Universal Robots PolyScope program: ratbit.urp

Program ratbit (installation=default directory=/programs createdIn=5.11.9.1010452 lastSavedIn=5.11.9.1010452 robotSerialNumber=20225200364)
Calibrated DH parameters: a=[0.00002, -0.569483, -0.54992, -0.00001, -0.000036, 0]; d=[0.180894, -146.691669, 192.918669, -46.053088, 0.119778, 0.115602]; alpha=[1.571425, -0.001534, 0.003359, 1.568739, -1.571477, 0]; deltaTheta=[0, 0.376258, -0.101074, -0.275185, -0.000002, 0]
Robot Program (runOnlyOnce=false)
  Script file /programs/Fuk_Rabbit_01D_newpath.script
    | def Machining1():
    |   # Global parameters:
    |   global speed_ms    = 0.300
    |   global speed_rads  = 0.750
    |   global accel_mss   = 3.000
    |   global accel_radss = 1.200
    |   global blend_radius_m = 0.001
    | 
    |   #--------------------------
    |   # Add any default subprograms here
    |   # For example, to drive a gripper as a program call:
    |   # def Gripper_Open():
    |   #   ...
    |   # end
    |   #
    |   # Example to drive a spray gun:
    |   def SprayOn(value):
    |     # use the value as an output:
    |     DO_SPRAY = 5
    |     if value == 0:
    |       set_standard_digital_out(DO_SPRAY, False)
    |     else:
    |       set_standard_digital_out(DO_SPRAY, True)
    |     end
    |   end
    |   #
    |   # Example to move an external axis
    |   def MoveAxis(value):
    |     # use the value as an output:
    |     DO_AXIS_1 = 1
    |     DI_AXIS_1 = 1
    |     if value <= 0:
    |       set_standard_digital_out(DO_AXIS_1, False)
    | 
    |       # Wait for digital input to change state
    |       #while (get_standard_digital_in(DI_AXIS_1) != False):
    |       #  sync()
    |       #end
    |     else:
    |       set_standard_digital_out(DO_AXIS_1, True)
    | 
    |       # Wait for digital input to change state
    |       #while (get_standard_digital_in(DI_AXIS_1) != True):
    |       #  sync()
    |       #end
    |     end
    |   end
    |   #--------------------------
    | 
    | 
    |   # Main program:
    |   # Program generated by RoboDK v5.4.3 for UR10e on 17/01/2023 09:30:10
    |   # Using nominal kinematics.
    |   blend_radius_m = 0.000
    |   speed_ms    = 1.000
    |   # set_reference(p[0.516600, -0.149080, 0.000000, 0.000000, 0.000000, 1.570796])
    |   set_tcp(p[0.000000, 0.000000, 0.25200, 0.000000, 0.000000, 0.000000])
    |   # Show Ballpen_2
    |   movej([0.053070, -1.824654, -1.998873, -4.030436, -1.570796, -1.517726],accel_radss,speed_rads,0,0)
    |   movel(p[0.486123, -0.148573, 0.015000, 0.000000, -3.141593, 0.000000],accel_mss,speed_ms,0,0)
    |   speed_ms    = 1.000
    |   movel(p[0.486123, -0.148573, 0.003000, 0.000000, -3.141593, 0.000000],accel_mss,speed_ms,0,blend_radius_m)
    |   speed_ms    = 0.050
    |   movel(p[0.486123, -0.148573, -0.000100, 0.000000, -3.141593, 0.000000],accel_mss,speed_ms,0,blend_radius_m)
    |   speed_ms    = 0.083
    |   movel(p[0.485906, -0.148799, -0.000100, 0.000000, -3.141593, 0.000000],accel_mss,speed_ms,0,0.000)
    |   movel(p[0.485689, -0.149025, -0.000100, 0.000000, -3.141593, 0.000000],accel_mss,speed_ms,0,0.000)
    |   movel(p[0.485511, -0.149199, -0.000100, 0.000000, -3.141593, 0.000000],accel_mss,speed_ms,0,0.000)
    |   movel(p[0.485335, -0.149346, -0.000100, 0.000000, -3.141593, 0.000000],accel_mss,speed_ms,0,0.000)
    |   movel(p[0.485182, -0.149454, -0.000100, 0.000000, -3.141593, 0.000000],accel_mss,speed_ms,0,0.000)
    |   movel(p[0.484988, -0.149437, -0.000100, 0.000000, -3.141593, 0.000000],accel_mss,speed_ms,0,0.000)
    |   movel(p[0.484142, -0.148632, -0.000100, 0.000000, -3.141593, 0.000000],accel_mss,speed_ms,0,blend_radius_m)
    |   movel(p[0.483183, -0.147699, -0.000100, 0.000000, -3.141593, 0.000000],accel_mss,speed_ms,0,blend_radius_m)
    |   movel(p[0.482074, -0.146592, -0.000100, 0.000000, -3.141593, 0.000000],accel_mss,speed_ms,0,blend_radius_m)
    |   movel(p[0.480976, -0.145473, -0.000100, 0.000000, -3.141593, 0.000000],accel_mss,speed_ms,0,blend_radius_m)
    |   movel(p[0.480046, -0.144505, -0.000100, 0.000000, -3.141593, 0.000000],accel_mss,speed_ms,0,blend_radius_m)
    |   movel(p[0.479240, -0.143652, -0.000100, 0.000000, -3.141593, 0.000000],accel_mss,speed_ms,0,blend_radius_m)
    |   movel(p[0.479187, -0.143544, -0.000100, 0.000000, -3.141593, 0.000000],accel_mss,speed_ms,0,0.000)
    |   movel(p[0.479279, -0.143263, -0.000100, 0.000000, -3.141593, 0.000000],accel_mss,speed_ms,0,0.000)
    |   movel(p[0.480734, -0.141843, -0.000100, 0.000000, -3.141593, 0.000000],accel_mss,speed_ms,0,blend_radius_m)
    |   movel(p[0.482145, -0.140509, -0.000100, 0.000000, -3.141593, 0.000000],accel_mss,speed_ms,0,blend_radius_m)
    |   movel(p[0.482666, -0.140186, -0.000100, 0.000000, -3.141593, 0.000000],accel_mss,speed_ms,0,blend_radius_m)
    |   movel(p[0.483571, -0.140040, -0.000100, 0.000000, -3.141593, 0.000000],accel_mss,speed_ms,0,blend_radius_m)
    |   movel(p[0.484504, -0.140251, -0.000100, 0.000000, -3.141593, 0.000000],accel_mss,speed_ms,0,blend_radius_m)
    |   movel(p[0.485320, -0.140784, -0.000100, 0.000000, -3.141593, 0.000000],accel_mss,speed_ms,0,blend_radius_m)
    |   movel(p[0.485889, -0.141559, -0.000100, 0.000000, -3.141593, 0.000000],accel_mss,speed_ms,0,blend_radius_m)
    |   movel(p[0.486167, -0.142427, -0.000100, 0.000000, -3.141593, 0.000000],accel_mss,speed_ms,0,blend_radius_m)
    |   movel(p[0.486122, -0.143201, -0.000100, 0.000000, -3.141593, 0.000000],accel_mss,speed_ms,0,blend_radius_m)
    |   movel(p[0.485720, -0.144015, -0.000100, 0.000000, -3.141593, 0.000000],accel_mss,speed_ms,0,blend_radius_m)
    |   movel(p[0.484872, -0.145041, -0.000100, 0.000000, -3.141593, 0.000000],accel_mss,speed_ms,0,blend_radius_m)
    |   movel(p[0.484523, -0.145430, -0.000100, 0.000000, -3.141593, 0.000000],accel_mss,speed_ms,0,blend_radius_m)
    |   movel(p[0.484229, -0.145788, -0.000100, 0.000000, -3.141593, 0.000000],accel_mss,speed_ms,0,0.000)
    |   movel(p[0.483998, -0.146094, -0.000100, 0.000000, -3.141593, 0.000000],accel_mss,speed_ms,0,0.000)
    |   movel(p[0.483961, -0.146209, -0.000100, 0.000000, -3.141593, 0.000000],accel_mss,speed_ms,0,0.000)
    |   movel(p[0.484001, -0.146324, -0.000100, 0.000000, -3.141593, 0.000000],accel_mss,speed_ms,0,0.000)
    |   movel(p[0.484278, -0.146661, -0.000100, 0.000000, -3.141593, 0.000000],accel_mss,speed_ms,0,0.000)
    |   movel(p[0.484628, -0.147054, -0.000100, 0.000000, -3.141593, 0.000000],accel_mss,speed_ms,0,blend_radius_m)
    |   movel(p[0.485042, -0.147484, -0.000100, 0.000000, -3.141593, 0.000000],accel_mss,speed_ms,0,blend_radius_m)
    |   movel(p[0.485582, -0.148028, -0.000100, 0.000000, -3.141593, 0.000000],accel_mss,speed_ms,0,blend_radius_m)
    |   movel(p[0.486123, -0.148573, -0.000100, 0.000000, -3.141593, 0.000000],accel_mss,speed_ms,0,blend_radius_m)
    |   speed_ms    = 0.050
    |   movel(p[0.486123, -0.148573, 0.003000, 0.000000, -3.141593, 0.000000],accel_mss,speed_ms,0,blend_radius_m)
    |   speed_ms    = 1.000
    |   movel(p[0.486123, -0.148573, 0.015000, 0.000000, -3.141593, 0.000000],accel_mss,speed_ms,0,blend_radius_m)
    |   movel(p[0.483124, -0.144911, 0.015000, 0.000000, -3.141593, 0.000000],accel_mss,speed_ms,0,blend_radius_m)
    |   movel(p[0.483124, -0.144911, 0.003000, 0.000000, -3.141593, 0.000000],accel_mss,speed_ms,0,blend_radius_m)
    |   speed_ms    = 0.050
    |   movel(p[0.483124, -0.144911, -0.000100, 0.000000, -3.141593, 0.000000],accel_mss,speed_ms,0,blend_radius_m)
    |   speed_ms    = 0.083
    |   movel(p[0.482775, -0.145021, -0.000100, 0.000000, -3.141593, 0.000000],accel_mss,speed_ms,0,0.000)
    |   movel(p[0.482418, -0.144857, -0.000100, 0.000000, -3.141593, 0.000000],accel_mss,speed_ms,0,0.000)
    |   movel(p[0.481726, -0.144152, -0.000100, 0.000000, -3.141593, 0.000000],accel_mss,speed_ms,0,blend_radius_m)
    |   movel(p[0.481290, -0.143631, -0.000100, 0.000000, -3.141593, 0.000000],accel_mss,speed_ms,0,blend_radius_m)
    |   movel(p[0.481235, -0.143353, -0.000100, 0.000000, -3.141593, 0.000000],accel_mss,speed_ms,0,0.000)
    |   movel(p[0.481407, -0.143059, -0.000100, 0.000000, -3.141593, 0.000000],accel_mss,speed_ms,0,0.000)
    |   movel(p[0.482217, -0.142290, -0.000100, 0.000000, -3.141593, 0.000000],accel_mss,speed_ms,0,blend_radius_m)
    |   movel(p[0.482465, -0.142075, -0.000100, 0.000000, -3.141593, 0.000000],accel_mss,speed_ms,0,0.000)
    |   movel(p[0.482730, -0.141875, -0.000100, 0.000000, -3.141593, 0.000000],accel_mss,speed_ms,0,0.000)
    |   movel(p[0.482975, -0.141713, -0.000100, 0.000000, -3.141593, 0.000000],accel_mss,speed_ms,0,0.000)
    |   movel(p[0.483149, -0.141630, -0.000100, 0.000000, -3.141593, 0.000000],accel_mss,speed_ms,0,0.000)
    |   movel(p[0.483717, -0.141623, -0.000100, 0.000000, -3.141593, 0.000000],accel_mss,speed_ms,0,blend_radius_m)
    |   movel(p[0.484256, -0.141955, -0.000100, 0.000000, -3.141593, 0.000000],accel_mss,speed_ms,0,blend_radius_m)
    |   movel(p[0.484596, -0.142514, -0.000100, 0.000000, -3.141593, 0.000000],accel_mss,speed_ms,0,blend_radius_m)
    |   movel(p[0.484618, -0.143123, -0.000100, 0.000000, -3.141593, 0.000000],accel_mss,speed_ms,0,blend_radius_m)
    |   movel(p[0.484529, -0.143332, -0.000100, 0.000000, -3.141593, 0.000000],accel_mss,speed_ms,0,0.000)
    |   movel(p[0.484314, -0.143650, -0.000100, 0.000000, -3.141593, 0.000000],accel_mss,speed_ms,0,0.000)
    |   movel(p[0.484037, -0.144003, -0.000100, 0.000000, -3.141593, 0.000000],accel_mss,speed_ms,0,0.000)
    |   movel(p[0.483729, -0.144344, -0.000100, 0.000000, -3.141593, 0.000000],accel_mss,speed_ms,0,0.000)
    |   movel(p[0.483124, -0.144911, -0.000100, 0.000000, -3.141593, 0.000000],accel_mss,speed_ms,0,blend_radius_m)
    |   speed_ms    = 0.050
    |   movel(p[0.483124, -0.144911, 0.003000, 0.000000, -3.141593, 0.000000],accel_mss,speed_ms,0,blend_radius_m)
    |   speed_ms    = 1.000
    |   movel(p[0.483124, -0.144911, 0.015000, 0.000000, -3.141593, 0.000000],accel_mss,speed_ms,0,blend_radius_m)
    |   movel(p[0.487811, -0.141414, 0.015000, 0.000000, -3.141593, 0.000000],accel_mss,speed_ms,0,blend_radius_m)
    |   movel(p[0.487811, -0.141414, 0.003000, 0.000000, -3.141593, 0.000000],accel_mss,speed_ms,0,blend_radius_m)
    |   speed_ms    = 0.050
    |   movel(p[0.487811, -0.141414, -0.000100, 0.000000, -3.141593, 0.000000],accel_mss,speed_ms,0,blend_radius_m)
    |   speed_ms    = 0.083
    |   movel(p[0.487491, -0.140892, -0.000100, 0.000000, -3.141593, 0.000000],accel_mss,speed_ms,0,blend_radius_m)
    |   movel(p[0.487400, -0.140626, -0.000100, 0.000000, -3.141593, 0.000000],accel_mss,speed_ms,0,0.000)
    |   movel(p[0.487339, -0.140285, -0.000100, 0.000000, -3.141593, 0.000000],accel_mss,speed_ms,0,0.000)
    |   movel(p[0.487307, -0.139892, -0.000100, 0.000000, -3.141593, 0.000000],accel_mss,speed_ms,0,0.000)
    |   movel(p[0.487310, -0.139469, -0.000100, 0.000000, -3.141593, 0.000000],accel_mss,speed_ms,0,0.000)
    |   movel(p[0.487439, -0.138661, -0.000100, 0.000000, -3.141593, 0.000000],accel_mss,speed_ms,0,blend_radius_m)
    |   movel(p[0.487749, -0.137963, -0.000100, 0.000000, -3.141593, 0.000000],accel_mss,speed_ms,0,blend_radius_m)
    |   movel(p[0.488242, -0.137381, -0.000100, 0.000000, -3.141593, 0.000000],accel_mss,speed_ms,0,blend_radius_m)
    |   movel(p[0.488911, -0.136916, -0.000100, 0.000000, -3.141593, 0.000000],accel_mss,speed_ms,0,blend_radius_m)
    |   movel(p[0.489677, -0.136642, -0.000100, 0.000000, -3.141593, 0.000000],accel_mss,speed_ms,0,blend_radius_m)
    |   movel(p[0.490526, -0.136585, -0.000100, 0.000000, -3.141593, 0.000000],accel_mss,speed_ms,0,blend_radius_m)
    |   movel(p[0.491362, -0.136747, -0.000100, 0.000000, -3.141593, 0.000000],accel_mss,speed_ms,0,blend_radius_m)
    |   movel(p[0.492092, -0.137115, -0.000100, 0.000000, -3.141593, 0.000000],accel_mss,speed_ms,0,blend_radius_m)
    |   movel(p[0.492654, -0.137612, -0.000100, 0.000000, -3.141593, 0.000000],accel_mss,speed_ms,0,blend_radius_m)
    |   movel(p[0.493144, -0.138258, -0.000100, 0.000000, -3.141593, 0.000000],accel_mss,speed_ms,0,blend_radius_m)
    |   movel(p[0.493503, -0.138962, -0.000100, 0.000000, -3.141593, 0.000000],accel_mss,speed_ms,0,blend_radius_m)
    |   movel(p[0.493671, -0.139629, -0.000100, 0.000000, -3.141593, 0.000000],accel_mss,speed_ms,0,blend_radius_m)
    |   movel(p[0.493430, -0.141150, -0.000100, 0.000000, -3.141593, 0.000000],accel_mss,speed_ms,0,blend_radius_m)
    |   movel(p[0.492438, -0.142384, -0.000100, 0.000000, -3.141593, 0.000000],accel_mss,speed_ms,0,blend_radius_m)
    |   movel(p[0.490977, -0.142992, -0.000100, 0.000000, -3.141593, 0.000000],accel_mss,speed_ms,0,blend_radius_m)
    |   movel(p[0.489451, -0.142800, -0.000100, 0.000000, -3.141593, 0.000000],accel_mss,speed_ms,0,blend_radius_m)
    |   movel(p[0.488923, -0.142496, -0.000100, 0.000000, -3.141593, 0.000000],accel_mss,speed_ms,0,blend_radius_m)
    |   movel(p[0.488334, -0.141990, -0.000100, 0.000000, -3.141593, 0.000000],accel_mss,speed_ms,0,blend_radius_m)
    |   movel(p[0.487811, -0.141414, -0.000100, 0.000000, -3.141593, 0.000000],accel_mss,speed_ms,0,blend_radius_m)
    |   speed_ms    = 0.050
    |   movel(p[0.487811, -0.141414, 0.003000, 0.000000, -3.141593, 0.000000],accel_mss,speed_ms,0,blend_radius_m)
    |   speed_ms    = 1.000
    |   movel(p[0.487811, -0.141414, 0.015000, 0.000000, -3.141593, 0.000000],accel_mss,speed_ms,0,blend_radius_m)
    |   movel(p[0.489267, -0.140905, 0.015000, 0.000000, -3.141593, 0.000000],accel_mss,speed_ms,0,blend_radius_m)
    |   movel(p[0.489267, -0.140905, 0.003000, 0.000000, -3.141593, 0.000000],accel_mss,speed_ms,0,blend_radius_m)
    |   speed_ms    = 0.050
    |   movel(p[0.489267, -0.140905, -0.000100, 0.000000, -3.141593, 0.000000],accel_mss,speed_ms,0,blend_radius_m)
    |   speed_ms    = 0.083
    |   movel(p[0.488764, -0.140201, -0.000100, 0.000000, -3.141593, 0.000000],accel_mss,speed_ms,0,blend_radius_m)
    |   movel(p[0.488534, -0.139500, -0.000100, 0.000000, -3.141593, 0.000000],accel_mss,speed_ms,0,blend_radius_m)
    |   movel(p[0.488593, -0.138851, -0.000100, 0.000000, -3.141593, 0.000000],accel_mss,speed_ms,0,blend_radius_m)
    |   movel(p[0.488924, -0.138290, -0.000100, 0.000000, -3.141593, 0.000000],accel_mss,speed_ms,0,blend_radius_m)
    |   movel(p[0.489534, -0.137898, -0.000100, 0.000000, -3.141593, 0.000000],accel_mss,speed_ms,0,blend_radius_m)
    |   movel(p[0.490256, -0.137841, -0.000100, 0.000000, -3.141593, 0.000000],accel_mss,speed_ms,0,blend_radius_m)
    |   movel(p[0.491020, -0.138140, -0.000100, 0.000000, -3.141593, 0.000000],accel_mss,speed_ms,0,blend_radius_m)
    |   movel(p[0.491739, -0.138764, -0.000100, 0.000000, -3.141593, 0.000000],accel_mss,speed_ms,0,blend_radius_m)
    |   movel(p[0.492146, -0.139301, -0.000100, 0.000000, -3.141593, 0.000000],accel_mss,speed_ms,0,blend_radius_m)
    |   movel(p[0.492374, -0.139794, -0.000100, 0.000000, -3.141593, 0.000000],accel_mss,speed_ms,0,blend_radius_m)
    |   movel(p[0.492436, -0.140272, -0.000100, 0.000000, -3.141593, 0.000000],accel_mss,speed_ms,0,0.000)
    |   movel(p[0.492345, -0.140761, -0.000100, 0.000000, -3.141593, 0.000000],accel_mss,speed_ms,0,0.000)
    |   movel(p[0.491847, -0.141407, -0.000100, 0.000000, -3.141593, 0.000000],accel_mss,speed_ms,0,blend_radius_m)
    |   movel(p[0.491027, -0.141679, -0.000100, 0.000000, -3.141593, 0.000000],accel_mss,speed_ms,0,blend_radius_m)
    |   movel(p[0.490083, -0.141499, -0.000100, 0.000000, -3.141593, 0.000000],accel_mss,speed_ms,0,blend_radius_m)
    |   movel(p[0.489267, -0.140905, -0.000100, 0.000000, -3.141593, 0.000000],accel_mss,speed_ms,0,blend_radius_m)
    |   speed_ms    = 0.050
    |   movel(p[0.489267, -0.140905, 0.003000, 0.000000, -3.141593, 0.000000],accel_mss,speed_ms,0,blend_radius_m)
    |   speed_ms    = 1.000
    |   movel(p[0.489267, -0.140905, 0.015000, 0.000000, -3.141593, 0.000000],accel_mss,speed_ms,0,blend_radius_m)
    |   movel(p[0.494074, -0.136704, 0.015000, 0.000000, -3.141593, 0.000000],accel_mss,speed_ms,0,blend_radius_m)
    |   movel(p[0.494074, -0.136704, 0.003000, 0.000000, -3.141593, 0.000000],accel_mss,speed_ms,0,blend_radius_m)
    |   speed_ms    = 0.050
    |   movel(p[0.494074, -0.136704, -0.000100, 0.000000, -3.141593, 0.000000],accel_mss,speed_ms,0,blend_radius_m)
    |   speed_ms    = 0.083
    |   movel(p[0.492928, -0.135570, -0.000100, 0.000000, -3.141593, 0.000000],accel_mss,speed_ms,0,blend_radius_m)
    |   movel(p[0.491447, -0.134091, -0.000100, 0.000000, -3.141593, 0.000000],accel_mss,speed_ms,0,blend_radius_m)
    |   movel(p[0.489967, -0.132612, -0.000100, 0.000000, -3.141593, 0.000000],accel_mss,speed_ms,0,blend_radius_m)
    |   movel(p[0.490207, -0.132364, -0.000100, 0.000000, -3.141593, 0.000000],accel_mss,speed_ms,0,0.000)
    |   movel(p[0.490447, -0.132117, -0.000100, 0.000000, -3.141593, 0.000000],accel_mss,speed_ms,0,0.000)
    |   movel(p[0.490686, -0.131869, -0.000100, 0.000000, -3.141593, 0.000000],accel_mss,speed_ms,0,0.000)
    |   movel(p[0.490926, -0.131622, -0.000100, 0.000000, -3.141593, 0.000000],accel_mss,speed_ms,0,0.000)
    |   movel(p[0.492410, -0.133104, -0.000100, 0.000000, -3.141593, 0.000000],accel_mss,speed_ms,0,blend_radius_m)
    |   movel(p[0.493894, -0.134586, -0.000100, 0.000000, -3.141593, 0.000000],accel_mss,speed_ms,0,blend_radius_m)
    |   movel(p[0.495031, -0.135733, -0.000100, 0.000000, -3.141593, 0.000000],accel_mss,speed_ms,0,blend_radius_m)
    |   movel(p[0.495989, -0.136721, -0.000100, 0.000000, -3.141593, 0.000000],accel_mss,speed_ms,0,blend_radius_m)
    |   movel(p[0.496823, -0.137596, -0.000100, 0.000000, -3.141593, 0.000000],accel_mss,speed_ms,0,blend_radius_m)
    |   movel(p[0.496861, -0.137692, -0.000100, 0.000000, -3.141593, 0.000000],accel_mss,speed_ms,0,0.000)
    |   movel(p[0.496796, -0.137879, -0.000100, 0.000000, -3.141593, 0.000000],accel_mss,speed_ms,0,0.000)
    |   movel(p[0.496527, -0.138185, -0.000100, 0.000000, -3.141593, 0.000000],accel_mss,speed_ms,0,0.000)
    |   movel(p[0.496230, -0.138462, -0.000100, 0.000000, -3.141593, 0.000000],accel_mss,speed_ms,0,0.000)
    |   movel(p[0.496049, -0.138528, -0.000100, 0.000000, -3.141593, 0.000000],accel_mss,speed_ms,0,0.000)
    |   movel(p[0.495941, -0.138486, -0.000100, 0.000000, -3.141593, 0.000000],accel_mss,speed_ms,0,0.000)
    |   movel(p[0.495066, -0.137659, -0.000100, 0.000000, -3.141593, 0.000000],accel_mss,speed_ms,0,blend_radius_m)
    |   movel(p[0.494074, -0.136704, -0.000100, 0.000000, -3.141593, 0.000000],accel_mss,speed_ms,0,blend_radius_m)
    |   speed_ms    = 0.050
    |   movel(p[0.494074, -0.136704, 0.003000, 0.000000, -3.141593, 0.000000],accel_mss,speed_ms,0,blend_radius_m)
    |   speed_ms    = 1.000
    |   movel(p[0.494074, -0.136704, 0.015000, 0.000000, -3.141593, 0.000000],accel_mss,speed_ms,0,blend_radius_m)
    |   movel(p[0.495341, -0.133290, 0.015000, 0.000000, -3.141593, 0.000000],accel_mss,speed_ms,0,blend_radius_m)
    |   movel(p[0.495341, -0.133290, 0.003000, 0.000000, -3.141593, 0.000000],accel_mss,speed_ms,0,blend_radius_m)
    |   speed_ms    = 0.050
    |   movel(p[0.495341, -0.133290, -0.000100, 0.000000, -3.141593, 0.000000],accel_mss,speed_ms,0,blend_radius_m)
    |   speed_ms    = 0.083
    |   movel(p[0.494409, -0.132847, -0.000100, 0.000000, -3.141593, 0.000000],accel_mss,speed_ms,0,blend_radius_m)
    |   movel(p[0.493590, -0.132450, -0.000100, 0.000000, -3.141593, 0.000000],accel_mss,speed_ms,0,blend_radius_m)
    |   movel(p[0.493631, -0.132230, -0.000100, 0.000000, -3.141593, 0.000000],accel_mss,speed_ms,0,0.000)
    |   movel(p[0.493992, -0.131876, -0.000100, 0.000000, -3.141593, 0.000000],accel_mss,speed_ms,0,blend_radius_m)
    |   movel(p[0.494374, -0.131546, -0.000100, 0.000000, -3.141593, 0.000000],accel_mss,speed_ms,0,blend_radius_m)
    |   movel(p[0.494564, -0.131478, -0.000100, 0.000000, -3.141593, 0.000000],accel_mss,speed_ms,0,0.000)
    |   movel(p[0.494698, -0.131507, -0.000100, 0.000000, -3.141593, 0.000000],accel_mss,speed_ms,0,0.000)
    |   movel(p[0.495213, -0.131743, -0.000100, 0.000000, -3.141593, 0.000000],accel_mss,speed_ms,0,blend_radius_m)
    |   movel(p[0.495818, -0.132033, -0.000100, 0.000000, -3.141593, 0.000000],accel_mss,speed_ms,0,blend_radius_m)
    |   movel(p[0.496498, -0.132378, -0.000100, 0.000000, -3.141593, 0.000000],accel_mss,speed_ms,0,blend_radius_m)
    |   movel(p[0.497622, -0.132946, -0.000100, 0.000000, -3.141593, 0.000000],accel_mss,speed_ms,0,blend_radius_m)
    |   movel(p[0.498224, -0.133197, -0.000100, 0.000000, -3.141593, 0.000000],accel_mss,speed_ms,0,blend_radius_m)
    |   movel(p[0.498543, -0.133247, -0.000100, 0.000000, -3.141593, 0.000000],accel_mss,speed_ms,0,0.000)
    |   movel(p[0.498661, -0.133126, -0.000100, 0.000000, -3.141593, 0.000000],accel_mss,speed_ms,0,0.000)
    |   movel(p[0.498637, -0.133018, -0.000100, 0.000000, -3.141593, 0.000000],accel_mss,speed_ms,0,0.000)
    |   movel(p[0.498377, -0.132453, -0.000100, 0.000000, -3.141593, 0.000000],accel_mss,speed_ms,0,blend_radius_m)
    |   movel(p[0.498065, -0.131796, -0.000100, 0.000000, -3.141593, 0.000000],accel_mss,speed_ms,0,blend_radius_m)
    |   movel(p[0.497695, -0.131047, -0.000100, 0.000000, -3.141593, 0.000000],accel_mss,speed_ms,0,blend_radius_m)
    |   movel(p[0.497212, -0.130083, -0.000100, 0.000000, -3.141593, 0.000000],accel_mss,speed_ms,0,blend_radius_m)
    |   movel(p[0.496729, -0.129119, -0.000100, 0.000000, -3.141593, 0.000000],accel_mss,speed_ms,0,blend_radius_m)
    |   movel(p[0.496985, -0.128871, -0.000100, 0.000000, -3.141593, 0.000000],accel_mss,speed_ms,0,0.000)
    |   movel(p[0.497241, -0.128624, -0.000100, 0.000000, -3.141593, 0.000000],accel_mss,speed_ms,0,0.000)
    |   movel(p[0.497497, -0.128376, -0.000100, 0.000000, -3.141593, 0.000000],accel_mss,speed_ms,0,0.000)
    |   movel(p[0.497752, -0.128128, -0.000100, 0.000000, -3.141593, 0.000000],accel_mss,speed_ms,0,0.000)
    |   movel(p[0.498286, -0.129247, -0.000100, 0.000000, -3.141593, 0.000000],accel_mss,speed_ms,0,blend_radius_m)
    |   movel(p[0.498819, -0.130366, -0.000100, 0.000000, -3.141593, 0.000000],accel_mss,speed_ms,0,blend_radius_m)
    |   # Splitting circular movement in 4 (instruction 203:MoveC 176)
    |   movel(p[0.499281, -0.131340, -0.000100, 0.000000, -3.141593, 0.000000],accel_mss,speed_ms,0,blend_radius_m)
    |   movel(p[0.499741, -0.132315, -0.000100, 0.000000, -3.141593, 0.000000],accel_mss,speed_ms,0,blend_radius_m)
    |   movel(p[0.500197, -0.133292, -0.000100, 0.000000, -3.141593, 0.000000],accel_mss,speed_ms,0,blend_radius_m)
    |   movel(p[0.500650, -0.134270, -0.000100, 0.000000, -3.141593, 0.000000],accel_mss,speed_ms,0,blend_radius_m)
    |   movel(p[0.501168, -0.135720, -0.000100, 0.000000, -3.141593, 0.000000],accel_mss,speed_ms,0,blend_radius_m)
    |   movel(p[0.501150, -0.136625, -0.000100, 0.000000, -3.141593, 0.000000],accel_mss,speed_ms,0,blend_radius_m)
    |   movel(p[0.500669, -0.137478, -0.000100, 0.000000, -3.141593, 0.000000],accel_mss,speed_ms,0,blend_radius_m)
    |   movel(p[0.500264, -0.137878, -0.000100, 0.000000, -3.141593, 0.000000],accel_mss,speed_ms,0,blend_radius_m)
    |   movel(p[0.499962, -0.138042, -0.000100, 0.000000, -3.141593, 0.000000],accel_mss,speed_ms,0,0.000)
    |   movel(p[0.499687, -0.138024, -0.000100, 0.000000, -3.141593, 0.000000],accel_mss,speed_ms,0,0.000)
    |   movel(p[0.499389, -0.137833, -0.000100, 0.000000, -3.141593, 0.000000],accel_mss,speed_ms,0,0.000)
    |   movel(p[0.499240, -0.137674, -0.000100, 0.000000, -3.141593, 0.000000],accel_mss,speed_ms,0,0.000)
    |   movel(p[0.499210, -0.137558, -0.000100, 0.000000, -3.141593, 0.000000],accel_mss,speed_ms,0,0.000)
    |   movel(p[0.499270, -0.137421, -0.000100, 0.000000, -3.141593, 0.000000],accel_mss,speed_ms,0,0.000)
    |   movel(p[0.499505, -0.137128, -0.000100, 0.000000, -3.141593, 0.000000],accel_mss,speed_ms,0,0.000)
    |   movel(p[0.499701, -0.136864, -0.000100, 0.000000, -3.141593, 0.000000],accel_mss,speed_ms,0,0.000)
    |   movel(p[0.499803, -0.136643, -0.000100, 0.000000, -3.141593, 0.000000],accel_mss,speed_ms,0,0.000)
    |   movel(p[0.499836, -0.136403, -0.000100, 0.000000, -3.141593, 0.000000],accel_mss,speed_ms,0,0.000)
    |   movel(p[0.499813, -0.136078, -0.000100, 0.000000, -3.141593, 0.000000],accel_mss,speed_ms,0,0.000)
    |   movel(p[0.499768, -0.135838, -0.000100, 0.000000, -3.141593, 0.000000],accel_mss,speed_ms,0,0.000)
    |   movel(p[0.499699, -0.135606, -0.000100, 0.000000, -3.141593, 0.000000],accel_mss,speed_ms,0,0.000)
    |   movel(p[0.499617, -0.135412, -0.000100, 0.000000, -3.141593, 0.000000],accel_mss,speed_ms,0,0.000)
    |   movel(p[0.499535, -0.135302, -0.000100, 0.000000, -3.141593, 0.000000],accel_mss,speed_ms,0,0.000)
    |   movel(p[0.499374, -0.135190, -0.000100, 0.000000, -3.141593, 0.000000],accel_mss,speed_ms,0,0.000)
    |   movel(p[0.498546, -0.134784, -0.000100, 0.000000, -3.141593, 0.000000],accel_mss,speed_ms,0,blend_radius_m)
    |   movel(p[0.497569, -0.134318, -0.000100, 0.000000, -3.141593, 0.000000],accel_mss,speed_ms,0,blend_radius_m)
    |   movel(p[0.496448, -0.133801, -0.000100, 0.000000, -3.141593, 0.000000],accel_mss,speed_ms,0,blend_radius_m)
    |   movel(p[0.495341, -0.133290, -0.000100, 0.000000, -3.141593, 0.000000],accel_mss,speed_ms,0,blend_radius_m)
    |   speed_ms    = 0.050
    |   movel(p[0.495341, -0.133290, 0.003000, 0.000000, -3.141593, 0.000000],accel_mss,speed_ms,0,blend_radius_m)
    |   speed_ms    = 1.000
    |   movel(p[0.495341, -0.133290, 0.015000, 0.000000, -3.141593, 0.000000],accel_mss,speed_ms,0,blend_radius_m)
    |   movel(p[0.500261, -0.128751, 0.015000, 0.000000, -3.141593, 0.000000],accel_mss,speed_ms,0,blend_radius_m)
    |   movel(p[0.500261, -0.128751, 0.003000, 0.000000, -3.141593, 0.000000],accel_mss,speed_ms,0,blend_radius_m)
    |   speed_ms    = 0.050
    |   movel(p[0.500261, -0.128751, -0.000100, 0.000000, -3.141593, 0.000000],accel_mss,speed_ms,0,blend_radius_m)
    |   speed_ms    = 0.083
    |   movel(p[0.499327, -0.127855, -0.000100, 0.000000, -3.141593, 0.000000],accel_mss,speed_ms,0,blend_radius_m)
    |   movel(p[0.498163, -0.126713, -0.000100, 0.000000, -3.141593, 0.000000],accel_mss,speed_ms,0,blend_radius_m)
    |   movel(p[0.497000, -0.125570, -0.000100, 0.000000, -3.141593, 0.000000],accel_mss,speed_ms,0,blend_radius_m)
    |   movel(p[0.497263, -0.125306, -0.000100, 0.000000, -3.141593, 0.000000],accel_mss,speed_ms,0,0.000)
    |   movel(p[0.497526, -0.125043, -0.000100, 0.000000, -3.141593, 0.000000],accel_mss,speed_ms,0,0.000)
    |   movel(p[0.497790, -0.124780, -0.000100, 0.000000, -3.141593, 0.000000],accel_mss,speed_ms,0,0.000)
    |   movel(p[0.498053, -0.124516, -0.000100, 0.000000, -3.141593, 0.000000],accel_mss,speed_ms,0,0.000)
    |   movel(p[0.499161, -0.125608, -0.000100, 0.000000, -3.141593, 0.000000],accel_mss,speed_ms,0,blend_radius_m)
    |   movel(p[0.500269, -0.126699, -0.000100, 0.000000, -3.141593, 0.000000],accel_mss,speed_ms,0,blend_radius_m)
    |   movel(p[0.501231, -0.127626, -0.000100, 0.000000, -3.141593, 0.000000],accel_mss,speed_ms,0,blend_radius_m)
    |   movel(p[0.502013, -0.128332, -0.000100, 0.000000, -3.141593, 0.000000],accel_mss,speed_ms,0,blend_radius_m)
    |   movel(p[0.502632, -0.128847, -0.000100, 0.000000, -3.141593, 0.000000],accel_mss,speed_ms,0,blend_radius_m)
    |   movel(p[0.502914, -0.128986, -0.000100, 0.000000, -3.141593, 0.000000],accel_mss,speed_ms,0,0.000)
    |   movel(p[0.503793, -0.128942, -0.000100, 0.000000, -3.141593, 0.000000],accel_mss,speed_ms,0,blend_radius_m)
    |   movel(p[0.504622, -0.128423, -0.000100, 0.000000, -3.141593, 0.000000],accel_mss,speed_ms,0,blend_radius_m)
    |   movel(p[0.505149, -0.127606, -0.000100, 0.000000, -3.141593, 0.000000],accel_mss,speed_ms,0,blend_radius_m)
    |   movel(p[0.505195, -0.126738, -0.000100, 0.000000, -3.141593, 0.000000],accel_mss,speed_ms,0,blend_radius_m)
    |   movel(p[0.505072, -0.126494, -0.000100, 0.000000, -3.141593, 0.000000],accel_mss,speed_ms,0,0.000)
    |   movel(p[0.504490, -0.125812, -0.000100, 0.000000, -3.141593, 0.000000],accel_mss,speed_ms,0,blend_radius_m)
    |   movel(p[0.503761, -0.125006, -0.000100, 0.000000, -3.141593, 0.000000],accel_mss,speed_ms,0,blend_radius_m)
    |   movel(p[0.502900, -0.124107, -0.000100, 0.000000, -3.141593, 0.000000],accel_mss,speed_ms,0,blend_radius_m)
    |   movel(p[0.501801, -0.122987, -0.000100, 0.000000, -3.141593, 0.000000],accel_mss,speed_ms,0,blend_radius_m)
    |   movel(p[0.500703, -0.121867, -0.000100, 0.000000, -3.141593, 0.000000],accel_mss,speed_ms,0,blend_radius_m)
    |   movel(p[0.500966, -0.121603, -0.000100, 0.000000, -3.141593, 0.000000],accel_mss,speed_ms,0,0.000)
    |   movel(p[0.501229, -0.121340, -0.000100, 0.000000, -3.141593, 0.000000],accel_mss,speed_ms,0,0.000)
    |   movel(p[0.501492, -0.121077, -0.000100, 0.000000, -3.141593, 0.000000],accel_mss,speed_ms,0,0.000)
    |   movel(p[0.501755, -0.120814, -0.000100, 0.000000, -3.141593, 0.000000],accel_mss,speed_ms,0,0.000)
    |   movel(p[0.502877, -0.121961, -0.000100, 0.000000, -3.141593, 0.000000],accel_mss,speed_ms,0,blend_radius_m)
    |   movel(p[0.503998, -0.123109, -0.000100, 0.000000, -3.141593, 0.000000],accel_mss,speed_ms,0,blend_radius_m)
    |   movel(p[0.504876, -0.124028, -0.000100, 0.000000, -3.141593, 0.000000],accel_mss,speed_ms,0,blend_radius_m)
    |   movel(p[0.505659, -0.124891, -0.000100, 0.000000, -3.141593, 0.000000],accel_mss,speed_ms,0,blend_radius_m)
    |   movel(p[0.506293, -0.125628, -0.000100, 0.000000, -3.141593, 0.000000],accel_mss,speed_ms,0,blend_radius_m)
    |   movel(p[0.506501, -0.125951, -0.000100, 0.000000, -3.141593, 0.000000],accel_mss,speed_ms,0,0.000)
    |   movel(p[0.506729, -0.126810, -0.000100, 0.000000, -3.141593, 0.000000],accel_mss,speed_ms,0,blend_radius_m)
    |   movel(p[0.506629, -0.127680, -0.000100, 0.000000, -3.141593, 0.000000],accel_mss,speed_ms,0,blend_radius_m)
    |   movel(p[0.506186, -0.128560, -0.000100, 0.000000, -3.141593, 0.000000],accel_mss,speed_ms,0,blend_radius_m)
    |   movel(p[0.505401, -0.129448, -0.000100, 0.000000, -3.141593, 0.000000],accel_mss,speed_ms,0,blend_radius_m)
    |   movel(p[0.504548, -0.130125, -0.000100, 0.000000, -3.141593, 0.000000],accel_mss,speed_ms,0,blend_radius_m)
    |   movel(p[0.503759, -0.130489, -0.000100, 0.000000, -3.141593, 0.000000],accel_mss,speed_ms,0,blend_radius_m)
    |   movel(p[0.502984, -0.130560, -0.000100, 0.000000, -3.141593, 0.000000],accel_mss,speed_ms,0,blend_radius_m)
    |   movel(p[0.502178, -0.130360, -0.000100, 0.000000, -3.141593, 0.000000],accel_mss,speed_ms,0,blend_radius_m)
    |   movel(p[0.501865, -0.130170, -0.000100, 0.000000, -3.141593, 0.000000],accel_mss,speed_ms,0,0.000)
    |   movel(p[0.501127, -0.129537, -0.000100, 0.000000, -3.141593, 0.000000],accel_mss,speed_ms,0,blend_radius_m)
    |   movel(p[0.500261, -0.128751, -0.000100, 0.000000, -3.141593, 0.000000],accel_mss,speed_ms,0,blend_radius_m)
    |   speed_ms    = 0.050
    |   movel(p[0.500261, -0.128751, 0.003000, 0.000000, -3.141593, 0.000000],accel_mss,speed_ms,0,blend_radius_m)
    |   speed_ms    = 1.000
    |   movel(p[0.500261, -0.128751, 0.015000, 0.000000, -3.141593, 0.000000],accel_mss,speed_ms,0,blend_radius_m)
    |   movel(p[0.508525, -0.119968, 0.015000, 0.000000, -3.141593, 0.000000],accel_mss,speed_ms,0,blend_radius_m)
    |   movel(p[0.508525, -0.119968, 0.003000, 0.000000, -3.141593, 0.000000],accel_mss,speed_ms,0,blend_radius_m)
    |   speed_ms    = 0.050
    |   movel(p[0.508525, -0.119968, -0.000100, 0.000000, -3.141593, 0.000000],accel_mss,speed_ms,0,blend_radius_m)
    |   speed_ms    = 0.083
    |   movel(p[0.507044, -0.118488, -0.000100, 0.000000, -3.141593, 0.000000],accel_mss,speed_ms,0,blend_radius_m)
    |   movel(p[0.505562, -0.117007, -0.000100, 0.000000, -3.141593, 0.000000],accel_mss,speed_ms,0,blend_radius_m)
    |   movel(p[0.505825, -0.116745, -0.000100, 0.000000, -3.141593, 0.000000],accel_mss,speed_ms,0,0.000)
    |   movel(p[0.506088, -0.116482, -0.000100, 0.000000, -3.141593, 0.000000],accel_mss,speed_ms,0,0.000)
    |   movel(p[0.506350, -0.116219, -0.000100, 0.000000, -3.141593, 0.000000],accel_mss,speed_ms,0,0.000)
    |   movel(p[0.506613, -0.115956, -0.000100, 0.000000, -3.141593, 0.000000],accel_mss,speed_ms,0,0.000)
    |   movel(p[0.508118, -0.117462, -0.000100, 0.000000, -3.141593, 0.000000],accel_mss,speed_ms,0,blend_radius_m)
    |   movel(p[0.509624, -0.118967, -0.000100, 0.000000, -3.141593, 0.000000],accel_mss,speed_ms,0,blend_radius_m)
    |   movel(p[0.511129, -0.120472, -0.000100, 0.000000, -3.141593, 0.000000],accel_mss,speed_ms,0,blend_radius_m)
    |   movel(p[0.512634, -0.121978, -0.000100, 0.000000, -3.141593, 0.000000],accel_mss,speed_ms,0,blend_radius_m)
    |   movel(p[0.512434, -0.122215, -0.000100, 0.000000, -3.141593, 0.000000],accel_mss,speed_ms,0,0.000)
    |   movel(p[0.512234, -0.122453, -0.000100, 0.000000, -3.141593, 0.000000],accel_mss,speed_ms,0,0.000)
    |   movel(p[0.512068, -0.122635, -0.000100, 0.000000, -3.141593, 0.000000],accel_mss,speed_ms,0,0.000)
    |   movel(p[0.511901, -0.122789, -0.000100, 0.000000, -3.141593, 0.000000],accel_mss,speed_ms,0,0.000)
    |   movel(p[0.511752, -0.122901, -0.000100, 0.000000, -3.141593, 0.000000],accel_mss,speed_ms,0,0.000)
    |   movel(p[0.511545, -0.122882, -0.000100, 0.000000, -3.141593, 0.000000],accel_mss,speed_ms,0,0.000)
    |   movel(p[0.510669, -0.122059, -0.000100, 0.000000, -3.141593, 0.000000],accel_mss,speed_ms,0,blend_radius_m)
    |   movel(p[0.509674, -0.121103, -0.000100, 0.000000, -3.141593, 0.000000],accel_mss,speed_ms,0,blend_radius_m)
    |   movel(p[0.508525, -0.119968, -0.000100, 0.000000, -3.141593, 0.000000],accel_mss,speed_ms,0,blend_radius_m)
    |   speed_ms    = 0.050
    |   movel(p[0.508525, -0.119968, 0.003000, 0.000000, -3.141593, 0.000000],accel_mss,speed_ms,0,blend_radius_m)
    |   speed_ms    = 1.000
    |   movel(p[0.508525, -0.119968, 0.015000, 0.000000, -3.141593, 0.000000],accel_mss,speed_ms,0,blend_radius_m)
    |   movel(p[0.510708, -0.117772, 0.015000, 0.000000, -3.141593, 0.000000],accel_mss,speed_ms,0,blend_radius_m)
    |   movel(p[0.510708, -0.117772, 0.003000, 0.000000, -3.141593, 0.000000],accel_mss,speed_ms,0,blend_radius_m)
    |   speed_ms    = 0.050
    |   movel(p[0.510708, -0.117772, -0.000100, 0.000000, -3.141593, 0.000000],accel_mss,speed_ms,0,blend_radius_m)
    |   speed_ms    = 0.083
    |   movel(p[0.510076, -0.117035, -0.000100, 0.000000, -3.141593, 0.000000],accel_mss,speed_ms,0,blend_radius_m)
    |   movel(p[0.509614, -0.116286, -0.000100, 0.000000, -3.141593, 0.000000],accel_mss,speed_ms,0,blend_radius_m)
    |   movel(p[0.509278, -0.115433, -0.000100, 0.000000, -3.141593, 0.000000],accel_mss,speed_ms,0,blend_radius_m)
    |   movel(p[0.509157, -0.114640, -0.000100, 0.000000, -3.141593, 0.000000],accel_mss,speed_ms,0,blend_radius_m)
    |   movel(p[0.509248, -0.113863, -0.000100, 0.000000, -3.141593, 0.000000],accel_mss,speed_ms,0,blend_radius_m)
    |   movel(p[0.509549, -0.113059, -0.000100, 0.000000, -3.141593, 0.000000],accel_mss,speed_ms,0,blend_radius_m)
    |   movel(p[0.510352, -0.111920, -0.000100, 0.000000, -3.141593, 0.000000],accel_mss,speed_ms,0,blend_radius_m)
    |   movel(p[0.511427, -0.111135, -0.000100, 0.000000, -3.141593, 0.000000],accel_mss,speed_ms,0,blend_radius_m)
    |   movel(p[0.512614, -0.110814, -0.000100, 0.000000, -3.141593, 0.000000],accel_mss,speed_ms,0,blend_radius_m)
    |   movel(p[0.513747, -0.110998, -0.000100, 0.000000, -3.141593, 0.000000],accel_mss,speed_ms,0,blend_radius_m)
    |   movel(p[0.514084, -0.111150, -0.000100, 0.000000, -3.141593, 0.000000],accel_mss,speed_ms,0,0.000)
    |   movel(p[0.514178, -0.111247, -0.000100, 0.000000, -3.141593, 0.000000],accel_mss,speed_ms,0,0.000)
    |   movel(p[0.514179, -0.111374, -0.000100, 0.000000, -3.141593, 0.000000],accel_mss,speed_ms,0,0.000)
    |   movel(p[0.514043, -0.111664, -0.000100, 0.000000, -3.141593, 0.000000],accel_mss,speed_ms,0,0.000)
    |   movel(p[0.513816, -0.112030, -0.000100, 0.000000, -3.141593, 0.000000],accel_mss,speed_ms,0,0.000)
    |   movel(p[0.513591, -0.112219, -0.000100, 0.000000, -3.141593, 0.000000],accel_mss,speed_ms,0,0.000)
    |   movel(p[0.513275, -0.112311, -0.000100, 0.000000, -3.141593, 0.000000],accel_mss,speed_ms,0,0.000)
    |   movel(p[0.512696, -0.112344, -0.000100, 0.000000, -3.141593, 0.000000],accel_mss,speed_ms,0,blend_radius_m)
    |   movel(p[0.512355, -0.112368, -0.000100, 0.000000, -3.141593, 0.000000],accel_mss,speed_ms,0,0.000)
    |   movel(p[0.512032, -0.112428, -0.000100, 0.000000, -3.141593, 0.000000],accel_mss,speed_ms,0,0.000)
    |   movel(p[0.511749, -0.112517, -0.000100, 0.000000, -3.141593, 0.000000],accel_mss,speed_ms,0,0.000)
    |   movel(p[0.511531, -0.112630, -0.000100, 0.000000, -3.141593, 0.000000],accel_mss,speed_ms,0,0.000)
    |   movel(p[0.511128, -0.113018, -0.000100, 0.000000, -3.141593, 0.000000],accel_mss,speed_ms,0,blend_radius_m)
    |   movel(p[0.510791, -0.113595, -0.000100, 0.000000, -3.141593, 0.000000],accel_mss,speed_ms,0,blend_radius_m)
    |   movel(p[0.510582, -0.114217, -0.000100, 0.000000, -3.141593, 0.000000],accel_mss,speed_ms,0,blend_radius_m)
    |   movel(p[0.510573, -0.114737, -0.000100, 0.000000, -3.141593, 0.000000],accel_mss,speed_ms,0,blend_radius_m)
    |   movel(p[0.510785, -0.115348, -0.000100, 0.000000, -3.141593, 0.000000],accel_mss,speed_ms,0,blend_radius_m)
    |   movel(p[0.511210, -0.116028, -0.000100, 0.000000, -3.141593, 0.000000],accel_mss,speed_ms,0,blend_radius_m)
    |   movel(p[0.511779, -0.116684, -0.000100, 0.000000, -3.141593, 0.000000],accel_mss,speed_ms,0,blend_radius_m)
    |   movel(p[0.512427, -0.117232, -0.000100, 0.000000, -3.141593, 0.000000],accel_mss,speed_ms,0,blend_radius_m)
    |   movel(p[0.512888, -0.117540, -0.000100, 0.000000, -3.141593, 0.000000],accel_mss,speed_ms,0,blend_radius_m)
    |   movel(p[0.513232, -0.117713, -0.000100, 0.000000, -3.141593, 0.000000],accel_mss,speed_ms,0,0.000)
    |   movel(p[0.513558, -0.117799, -0.000100, 0.000000, -3.141593, 0.000000],accel_mss,speed_ms,0,0.000)
    |   movel(p[0.513948, -0.117828, -0.000100, 0.000000, -3.141593, 0.000000],accel_mss,speed_ms,0,0.000)
    |   movel(p[0.514831, -0.117665, -0.000100, 0.000000, -3.141593, 0.000000],accel_mss,speed_ms,0,blend_radius_m)
    |   movel(p[0.515531, -0.117201, -0.000100, 0.000000, -3.141593, 0.000000],accel_mss,speed_ms,0,blend_radius_m)
    |   movel(p[0.515944, -0.116501, -0.000100, 0.000000, -3.141593, 0.000000],accel_mss,speed_ms,0,blend_radius_m)
    |   movel(p[0.516019, -0.115666, -0.000100, 0.000000, -3.141593, 0.000000],accel_mss,speed_ms,0,blend_radius_m)
    |   movel(p[0.515983, -0.115414, -0.000100, 0.000000, -3.141593, 0.000000],accel_mss,speed_ms,0,0.000)
    |   movel(p[0.515938, -0.115165, -0.000100, 0.000000, -3.141593, 0.000000],accel_mss,speed_ms,0,0.000)
    |   movel(p[0.515890, -0.114949, -0.000100, 0.000000, -3.141593, 0.000000],accel_mss,speed_ms,0,0.000)
    |   movel(p[0.515848, -0.114821, -0.000100, 0.000000, -3.141593, 0.000000],accel_mss,speed_ms,0,0.000)
    |   movel(p[0.515838, -0.114700, -0.000100, 0.000000, -3.141593, 0.000000],accel_mss,speed_ms,0,0.000)
    |   movel(p[0.515899, -0.114583, -0.000100, 0.000000, -3.141593, 0.000000],accel_mss,speed_ms,0,0.000)
    |   movel(p[0.516043, -0.114464, -0.000100, 0.000000, -3.141593, 0.000000],accel_mss,speed_ms,0,0.000)
    |   movel(p[0.516286, -0.114333, -0.000100, 0.000000, -3.141593, 0.000000],accel_mss,speed_ms,0,0.000)
    |   movel(p[0.516787, -0.114123, -0.000100, 0.000000, -3.141593, 0.000000],accel_mss,speed_ms,0,blend_radius_m)
    |   movel(p[0.517051, -0.114115, -0.000100, 0.000000, -3.141593, 0.000000],accel_mss,speed_ms,0,0.000)
    |   movel(p[0.517232, -0.114266, -0.000100, 0.000000, -3.141593, 0.000000],accel_mss,speed_ms,0,0.000)
    |   movel(p[0.517387, -0.114658, -0.000100, 0.000000, -3.141593, 0.000000],accel_mss,speed_ms,0,0.000)
    |   movel(p[0.517554, -0.115572, -0.000100, 0.000000, -3.141593, 0.000000],accel_mss,speed_ms,0,blend_radius_m)
    |   movel(p[0.517483, -0.116398, -0.000100, 0.000000, -3.141593, 0.000000],accel_mss,speed_ms,0,blend_radius_m)
    |   movel(p[0.517160, -0.117181, -0.000100, 0.000000, -3.141593, 0.000000],accel_mss,speed_ms,0,blend_radius_m)
    |   movel(p[0.516573, -0.117973, -0.000100, 0.000000, -3.141593, 0.000000],accel_mss,speed_ms,0,blend_radius_m)
    |   movel(p[0.515947, -0.118564, -0.000100, 0.000000, -3.141593, 0.000000],accel_mss,speed_ms,0,blend_radius_m)
    |   movel(p[0.515320, -0.118953, -0.000100, 0.000000, -3.141593, 0.000000],accel_mss,speed_ms,0,blend_radius_m)
    |   movel(p[0.514628, -0.119170, -0.000100, 0.000000, -3.141593, 0.000000],accel_mss,speed_ms,0,blend_radius_m)
    |   movel(p[0.513811, -0.119242, -0.000100, 0.000000, -3.141593, 0.000000],accel_mss,speed_ms,0,blend_radius_m)
    |   movel(p[0.513311, -0.119224, -0.000100, 0.000000, -3.141593, 0.000000],accel_mss,speed_ms,0,blend_radius_m)
    |   movel(p[0.512906, -0.119166, -0.000100, 0.000000, -3.141593, 0.000000],accel_mss,speed_ms,0,0.000)
    |   movel(p[0.512544, -0.119061, -0.000100, 0.000000, -3.141593, 0.000000],accel_mss,speed_ms,0,0.000)
    |   movel(p[0.512177, -0.118896, -0.000100, 0.000000, -3.141593, 0.000000],accel_mss,speed_ms,0,0.000)
    |   movel(p[0.511434, -0.118418, -0.000100, 0.000000, -3.141593, 0.000000],accel_mss,speed_ms,0,blend_radius_m)
    |   movel(p[0.510708, -0.117772, -0.000100, 0.000000, -3.141593, 0.000000],accel_mss,speed_ms,0,blend_radius_m)
    |   speed_ms    = 0.050
    |   movel(p[0.510708, -0.117772, 0.003000, 0.000000, -3.141593, 0.000000],accel_mss,speed_ms,0,blend_radius_m)
    |   speed_ms    = 1.000
    |   movel(p[0.510708, -0.117772, 0.015000, 0.000000, -3.141593, 0.000000],accel_mss,speed_ms,0,blend_radius_m)
    |   movel(p[0.495781, -0.118072, 0.015000, 0.000000, -3.141593, 0.000000],accel_mss,speed_ms,0,blend_radius_m)
    |   movel(p[0.495781, -0.118072, 0.003000, 0.000000, -3.141593, 0.000000],accel_mss,speed_ms,0,blend_radius_m)
    |   speed_ms    = 0.050
    |   movel(p[0.495781, -0.118072, -0.000100, 0.000000, -3.141593, 0.000000],accel_mss,speed_ms,0,blend_radius_m)
    |   speed_ms    = 0.083
    |   movel(p[0.495758, -0.120763, -0.000100, 0.000000, -3.141593, 0.000000],accel_mss,speed_ms,0,blend_radius_m)
    |   movel(p[0.495736, -0.123453, -0.000100, 0.000000, -3.141593, 0.000000],accel_mss,speed_ms,0,blend_radius_m)
    |   movel(p[0.495511, -0.123860, -0.000100, 0.000000, -3.141593, 0.000000],accel_mss,speed_ms,0,0.000)
    |   movel(p[0.495286, -0.124266, -0.000100, 0.000000, -3.141593, 0.000000],accel_mss,speed_ms,0,0.000)
    |   movel(p[0.493952, -0.125719, -0.000100, 0.000000, -3.141593, 0.000000],accel_mss,speed_ms,0,blend_radius_m)
    |   movel(p[0.492074, -0.126439, -0.000100, 0.000000, -3.141593, 0.000000],accel_mss,speed_ms,0,blend_radius_m)
    |   movel(p[0.490072, -0.126271, -0.000100, 0.000000, -3.141593, 0.000000],accel_mss,speed_ms,0,blend_radius_m)
    |   movel(p[0.488391, -0.125248, -0.000100, 0.000000, -3.141593, 0.000000],accel_mss,speed_ms,0,blend_radius_m)
    |   movel(p[0.487830, -0.124563, -0.000100, 0.000000, -3.141593, 0.000000],accel_mss,speed_ms,0,blend_radius_m)
    |   movel(p[0.487455, -0.123823, -0.000100, 0.000000, -3.141593, 0.000000],accel_mss,speed_ms,0,blend_radius_m)
    |   movel(p[0.487227, -0.122920, -0.000100, 0.000000, -3.141593, 0.000000],accel_mss,speed_ms,0,blend_radius_m)
    |   movel(p[0.487112, -0.121728, -0.000100, 0.000000, -3.141593, 0.000000],accel_mss,speed_ms,0,blend_radius_m)
    |   movel(p[0.487074, -0.120941, -0.000100, 0.000000, -3.141593, 0.000000],accel_mss,speed_ms,0,blend_radius_m)
    |   movel(p[0.487036, -0.120153, -0.000100, 0.000000, -3.141593, 0.000000],accel_mss,speed_ms,0,blend_radius_m)
    |   movel(p[0.486305, -0.120132, -0.000100, 0.000000, -3.141593, 0.000000],accel_mss,speed_ms,0,blend_radius_m)
    |   movel(p[0.485573, -0.120110, -0.000100, 0.000000, -3.141593, 0.000000],accel_mss,speed_ms,0,blend_radius_m)
    |   movel(p[0.484842, -0.120089, -0.000100, 0.000000, -3.141593, 0.000000],accel_mss,speed_ms,0,blend_radius_m)
    |   movel(p[0.484111, -0.120067, -0.000100, 0.000000, -3.141593, 0.000000],accel_mss,speed_ms,0,blend_radius_m)
    |   movel(p[0.484111, -0.119508, -0.000100, 0.000000, -3.141593, 0.000000],accel_mss,speed_ms,0,blend_radius_m)
    |   movel(p[0.484111, -0.118948, -0.000100, 0.000000, -3.141593, 0.000000],accel_mss,speed_ms,0,blend_radius_m)
    |   movel(p[0.484111, -0.118388, -0.000100, 0.000000, -3.141593, 0.000000],accel_mss,speed_ms,0,blend_radius_m)
    |   movel(p[0.484111, -0.117828, -0.000100, 0.000000, -3.141593, 0.000000],accel_mss,speed_ms,0,blend_radius_m)
    |   movel(p[0.486177, -0.117828, -0.000100, 0.000000, -3.141593, 0.000000],accel_mss,speed_ms,0,blend_radius_m)
    |   movel(p[0.488243, -0.117828, -0.000100, 0.000000, -3.141593, 0.000000],accel_mss,speed_ms,0,blend_radius_m)
    |   movel(p[0.490308, -0.117828, -0.000100, 0.000000, -3.141593, 0.000000],accel_mss,speed_ms,0,blend_radius_m)
    |   movel(p[0.492374, -0.117828, -0.000100, 0.000000, -3.141593, 0.000000],accel_mss,speed_ms,0,blend_radius_m)
    |   movel(p[0.492352, -0.118372, -0.000100, 0.000000, -3.141593, 0.000000],accel_mss,speed_ms,0,blend_radius_m)
    |   movel(p[0.492330, -0.118916, -0.000100, 0.000000, -3.141593, 0.000000],accel_mss,speed_ms,0,blend_radius_m)
    |   movel(p[0.492308, -0.119460, -0.000100, 0.000000, -3.141593, 0.000000],accel_mss,speed_ms,0,blend_radius_m)
    |   movel(p[0.492286, -0.120003, -0.000100, 0.000000, -3.141593, 0.000000],accel_mss,speed_ms,0,blend_radius_m)
    |   movel(p[0.491548, -0.120025, -0.000100, 0.000000, -3.141593, 0.000000],accel_mss,speed_ms,0,blend_radius_m)
    |   movel(p[0.490810, -0.120046, -0.000100, 0.000000, -3.141593, 0.000000],accel_mss,speed_ms,0,blend_radius_m)
    |   movel(p[0.490071, -0.120068, -0.000100, 0.000000, -3.141593, 0.000000],accel_mss,speed_ms,0,blend_radius_m)
    |   movel(p[0.489333, -0.120090, -0.000100, 0.000000, -3.141593, 0.000000],accel_mss,speed_ms,0,blend_radius_m)
    |   movel(p[0.489359, -0.120831, -0.000100, 0.000000, -3.141593, 0.000000],accel_mss,speed_ms,0,blend_radius_m)
    |   movel(p[0.489385, -0.121572, -0.000100, 0.000000, -3.141593, 0.000000],accel_mss,speed_ms,0,blend_radius_m)
    |   movel(p[0.489426, -0.122441, -0.000100, 0.000000, -3.141593, 0.000000],accel_mss,speed_ms,0,blend_radius_m)
    |   movel(p[0.489488, -0.122880, -0.000100, 0.000000, -3.141593, 0.000000],accel_mss,speed_ms,0,0.000)
    |   movel(p[0.489604, -0.123176, -0.000100, 0.000000, -3.141593, 0.000000],accel_mss,speed_ms,0,0.000)
    |   movel(p[0.489811, -0.123456, -0.000100, 0.000000, -3.141593, 0.000000],accel_mss,speed_ms,0,0.000)
    |   movel(p[0.490694, -0.124082, -0.000100, 0.000000, -3.141593, 0.000000],accel_mss,speed_ms,0,blend_radius_m)
    |   movel(p[0.491696, -0.124256, -0.000100, 0.000000, -3.141593, 0.000000],accel_mss,speed_ms,0,blend_radius_m)
    |   movel(p[0.492632, -0.123945, -0.000100, 0.000000, -3.141593, 0.000000],accel_mss,speed_ms,0,blend_radius_m)
    |   movel(p[0.493336, -0.123211, -0.000100, 0.000000, -3.141593, 0.000000],accel_mss,speed_ms,0,blend_radius_m)
    |   movel(p[0.493507, -0.122770, -0.000100, 0.000000, -3.141593, 0.000000],accel_mss,speed_ms,0,0.000)
    |   movel(p[0.493597, -0.122132, -0.000100, 0.000000, -3.141593, 0.000000],accel_mss,speed_ms,0,blend_radius_m)
    |   movel(p[0.493647, -0.121029, -0.000100, 0.000000, -3.141593, 0.000000],accel_mss,speed_ms,0,blend_radius_m)
    |   movel(p[0.493682, -0.118459, -0.000100, 0.000000, -3.141593, 0.000000],accel_mss,speed_ms,0,blend_radius_m)
    |   movel(p[0.493718, -0.115658, -0.000100, 0.000000, -3.141593, 0.000000],accel_mss,speed_ms,0,blend_radius_m)
    |   movel(p[0.493764, -0.114742, -0.000100, 0.000000, -3.141593, 0.000000],accel_mss,speed_ms,0,blend_radius_m)
    |   movel(p[0.493859, -0.114293, -0.000100, 0.000000, -3.141593, 0.000000],accel_mss,speed_ms,0,0.000)
    |   movel(p[0.494057, -0.114088, -0.000100, 0.000000, -3.141593, 0.000000],accel_mss,speed_ms,0,0.000)
    |   movel(p[0.494229, -0.114000, -0.000100, 0.000000, -3.141593, 0.000000],accel_mss,speed_ms,0,0.000)
    |   movel(p[0.494501, -0.113812, -0.000100, 0.000000, -3.141593, 0.000000],accel_mss,speed_ms,0,0.000)
    |   movel(p[0.494806, -0.113578, -0.000100, 0.000000, -3.141593, 0.000000],accel_mss,speed_ms,0,0.000)
    |   movel(p[0.495106, -0.113326, -0.000100, 0.000000, -3.141593, 0.000000],accel_mss,speed_ms,0,0.000)
    |   movel(p[0.495465, -0.113008, -0.000100, 0.000000, -3.141593, 0.000000],accel_mss,speed_ms,0,0.000)
    |   movel(p[0.495825, -0.112690, -0.000100, 0.000000, -3.141593, 0.000000],accel_mss,speed_ms,0,0.000)
    |   movel(p[0.495803, -0.115381, -0.000100, 0.000000, -3.141593, 0.000000],accel_mss,speed_ms,0,blend_radius_m)
    |   movel(p[0.495781, -0.118072, -0.000100, 0.000000, -3.141593, 0.000000],accel_mss,speed_ms,0,blend_radius_m)
    |   speed_ms    = 0.050
    |   movel(p[0.495781, -0.118072, 0.003000, 0.000000, -3.141593, 0.000000],accel_mss,speed_ms,0,blend_radius_m)
    |   speed_ms    = 1.000
    |   movel(p[0.495781, -0.118072, 0.015000, 0.000000, -3.141593, 0.000000],accel_mss,speed_ms,0,blend_radius_m)
    |   movel(p[0.486582, -0.124567, 0.015000, 0.000000, -3.141593, 0.000000],accel_mss,speed_ms,0,blend_radius_m)
    |   movel(p[0.486582, -0.124567, 0.003000, 0.000000, -3.141593, 0.000000],accel_mss,speed_ms,0,blend_radius_m)
    |   speed_ms    = 0.050
    |   movel(p[0.486582, -0.124567, -0.000100, 0.000000, -3.141593, 0.000000],accel_mss,speed_ms,0,blend_radius_m)
    |   speed_ms    = 0.083
    |   movel(p[0.486660, -0.124735, -0.000100, 0.000000, -3.141593, 0.000000],accel_mss,speed_ms,0,0.000)
    |   movel(p[0.486851, -0.125029, -0.000100, 0.000000, -3.141593, 0.000000],accel_mss,speed_ms,0,0.000)
    |   movel(p[0.487092, -0.125366, -0.000100, 0.000000, -3.141593, 0.000000],accel_mss,speed_ms,0,0.000)
    |   movel(p[0.487359, -0.125708, -0.000100, 0.000000, -3.141593, 0.000000],accel_mss,speed_ms,0,0.000)
    |   movel(p[0.487699, -0.126126, -0.000100, 0.000000, -3.141593, 0.000000],accel_mss,speed_ms,0,blend_radius_m)
    |   movel(p[0.488039, -0.126543, -0.000100, 0.000000, -3.141593, 0.000000],accel_mss,speed_ms,0,blend_radius_m)
    |   movel(p[0.485388, -0.126520, -0.000100, 0.000000, -3.141593, 0.000000],accel_mss,speed_ms,0,blend_radius_m)
    |   movel(p[0.482738, -0.126498, -0.000100, 0.000000, -3.141593, 0.000000],accel_mss,speed_ms,0,blend_radius_m)
    |   movel(p[0.479275, -0.126462, -0.000100, 0.000000, -3.141593, 0.000000],accel_mss,speed_ms,0,blend_radius_m)
    |   movel(p[0.478035, -0.126413, -0.000100, 0.000000, -3.141593, 0.000000],accel_mss,speed_ms,0,blend_radius_m)
    |   movel(p[0.477329, -0.126310, -0.000100, 0.000000, -3.141593, 0.000000],accel_mss,speed_ms,0,blend_radius_m)
    |   movel(p[0.476761, -0.126100, -0.000100, 0.000000, -3.141593, 0.000000],accel_mss,speed_ms,0,blend_radius_m)
    |   movel(p[0.475900, -0.125540, -0.000100, 0.000000, -3.141593, 0.000000],accel_mss,speed_ms,0,blend_radius_m)
    |   movel(p[0.475213, -0.124857, -0.000100, 0.000000, -3.141593, 0.000000],accel_mss,speed_ms,0,blend_radius_m)
    |   movel(p[0.474703, -0.124049, -0.000100, 0.000000, -3.141593, 0.000000],accel_mss,speed_ms,0,blend_radius_m)
    |   movel(p[0.474366, -0.123118, -0.000100, 0.000000, -3.141593, 0.000000],accel_mss,speed_ms,0,blend_radius_m)
    |   movel(p[0.474266, -0.122037, -0.000100, 0.000000, -3.141593, 0.000000],accel_mss,speed_ms,0,blend_radius_m)
    |   movel(p[0.474480, -0.120903, -0.000100, 0.000000, -3.141593, 0.000000],accel_mss,speed_ms,0,blend_radius_m)
    |   movel(p[0.474980, -0.119840, -0.000100, 0.000000, -3.141593, 0.000000],accel_mss,speed_ms,0,blend_radius_m)
    |   movel(p[0.475716, -0.118967, -0.000100, 0.000000, -3.141593, 0.000000],accel_mss,speed_ms,0,blend_radius_m)
    |   movel(p[0.476395, -0.118440, -0.000100, 0.000000, -3.141593, 0.000000],accel_mss,speed_ms,0,blend_radius_m)
    |   movel(p[0.477042, -0.118122, -0.000100, 0.000000, -3.141593, 0.000000],accel_mss,speed_ms,0,blend_radius_m)
    |   movel(p[0.477835, -0.117939, -0.000100, 0.000000, -3.141593, 0.000000],accel_mss,speed_ms,0,blend_radius_m)
    |   movel(p[0.479011, -0.117836, -0.000100, 0.000000, -3.141593, 0.000000],accel_mss,speed_ms,0,blend_radius_m)
    |   movel(p[0.479798, -0.117794, -0.000100, 0.000000, -3.141593, 0.000000],accel_mss,speed_ms,0,blend_radius_m)
    |   movel(p[0.480586, -0.117753, -0.000100, 0.000000, -3.141593, 0.000000],accel_mss,speed_ms,0,blend_radius_m)
    |   movel(p[0.480604, -0.117491, -0.000100, 0.000000, -3.141593, 0.000000],accel_mss,speed_ms,0,0.000)
    |   movel(p[0.480623, -0.117228, -0.000100, 0.000000, -3.141593, 0.000000],accel_mss,speed_ms,0,0.000)
    |   movel(p[0.480643, -0.116963, -0.000100, 0.000000, -3.141593, 0.000000],accel_mss,speed_ms,0,0.000)
    |   movel(p[0.480675, -0.116580, -0.000100, 0.000000, -3.141593, 0.000000],accel_mss,speed_ms,0,0.000)
    |   movel(p[0.480712, -0.116159, -0.000100, 0.000000, -3.141593, 0.000000],accel_mss,speed_ms,0,0.000)
    |   movel(p[0.480748, -0.115760, -0.000100, 0.000000, -3.141593, 0.000000],accel_mss,speed_ms,0,0.000)
    |   movel(p[0.480792, -0.115288, -0.000100, 0.000000, -3.141593, 0.000000],accel_mss,speed_ms,0,0.000)
    |   movel(p[0.480836, -0.114816, -0.000100, 0.000000, -3.141593, 0.000000],accel_mss,speed_ms,0,0.000)
    |   movel(p[0.481374, -0.114838, -0.000100, 0.000000, -3.141593, 0.000000],accel_mss,speed_ms,0,blend_radius_m)
    |   movel(p[0.481911, -0.114860, -0.000100, 0.000000, -3.141593, 0.000000],accel_mss,speed_ms,0,blend_radius_m)
    |   movel(p[0.482449, -0.114881, -0.000100, 0.000000, -3.141593, 0.000000],accel_mss,speed_ms,0,blend_radius_m)
    |   movel(p[0.482986, -0.114903, -0.000100, 0.000000, -3.141593, 0.000000],accel_mss,speed_ms,0,blend_radius_m)
    |   movel(p[0.483007, -0.116778, -0.000100, 0.000000, -3.141593, 0.000000],accel_mss,speed_ms,0,blend_radius_m)
    |   movel(p[0.483028, -0.118653, -0.000100, 0.000000, -3.141593, 0.000000],accel_mss,speed_ms,0,blend_radius_m)
    |   movel(p[0.483038, -0.120115, -0.000100, 0.000000, -3.141593, 0.000000],accel_mss,speed_ms,0,blend_radius_m)
    |   movel(p[0.483033, -0.121403, -0.000100, 0.000000, -3.141593, 0.000000],accel_mss,speed_ms,0,blend_radius_m)
    |   movel(p[0.483019, -0.122496, -0.000100, 0.000000, -3.141593, 0.000000],accel_mss,speed_ms,0,blend_radius_m)
    |   movel(p[0.482986, -0.122747, -0.000100, 0.000000, -3.141593, 0.000000],accel_mss,speed_ms,0,0.000)
    |   movel(p[0.482897, -0.122938, -0.000100, 0.000000, -3.141593, 0.000000],accel_mss,speed_ms,0,0.000)
    |   movel(p[0.482756, -0.123035, -0.000100, 0.000000, -3.141593, 0.000000],accel_mss,speed_ms,0,0.000)
    |   movel(p[0.482488, -0.123066, -0.000100, 0.000000, -3.141593, 0.000000],accel_mss,speed_ms,0,0.000)
    |   movel(p[0.481819, -0.123047, -0.000100, 0.000000, -3.141593, 0.000000],accel_mss,speed_ms,0,blend_radius_m)
    |   movel(p[0.481277, -0.123025, -0.000100, 0.000000, -3.141593, 0.000000],accel_mss,speed_ms,0,blend_radius_m)
    |   movel(p[0.480736, -0.123003, -0.000100, 0.000000, -3.141593, 0.000000],accel_mss,speed_ms,0,blend_radius_m)
    |   movel(p[0.480714, -0.122265, -0.000100, 0.000000, -3.141593, 0.000000],accel_mss,speed_ms,0,blend_radius_m)
    |   movel(p[0.480693, -0.121527, -0.000100, 0.000000, -3.141593, 0.000000],accel_mss,speed_ms,0,blend_radius_m)
    |   movel(p[0.480671, -0.120789, -0.000100, 0.000000, -3.141593, 0.000000],accel_mss,speed_ms,0,blend_radius_m)
    |   movel(p[0.480650, -0.120051, -0.000100, 0.000000, -3.141593, 0.000000],accel_mss,speed_ms,0,blend_radius_m)
    |   movel(p[0.479907, -0.120076, -0.000100, 0.000000, -3.141593, 0.000000],accel_mss,speed_ms,0,blend_radius_m)
    |   movel(p[0.479165, -0.120102, -0.000100, 0.000000, -3.141593, 0.000000],accel_mss,speed_ms,0,blend_radius_m)
    |   movel(p[0.478251, -0.120145, -0.000100, 0.000000, -3.141593, 0.000000],accel_mss,speed_ms,0,blend_radius_m)
    |   movel(p[0.477830, -0.120210, -0.000100, 0.000000, -3.141593, 0.000000],accel_mss,speed_ms,0,0.000)
    |   movel(p[0.477537, -0.120339, -0.000100, 0.000000, -3.141593, 0.000000],accel_mss,speed_ms,0,0.000)
    |   movel(p[0.477224, -0.120591, -0.000100, 0.000000, -3.141593, 0.000000],accel_mss,speed_ms,0,0.000)
    |   movel(p[0.476720, -0.121271, -0.000100, 0.000000, -3.141593, 0.000000],accel_mss,speed_ms,0,blend_radius_m)
    |   movel(p[0.476507, -0.122043, -0.000100, 0.000000, -3.141593, 0.000000],accel_mss,speed_ms,0,blend_radius_m)
    |   movel(p[0.476611, -0.122825, -0.000100, 0.000000, -3.141593, 0.000000],accel_mss,speed_ms,0,blend_radius_m)
    |   movel(p[0.477016, -0.123537, -0.000100, 0.000000, -3.141593, 0.000000],accel_mss,speed_ms,0,blend_radius_m)
    |   movel(p[0.477195, -0.123727, -0.000100, 0.000000, -3.141593, 0.000000],accel_mss,speed_ms,0,0.000)
    |   movel(p[0.477408, -0.123912, -0.000100, 0.000000, -3.141593, 0.000000],accel_mss,speed_ms,0,0.000)
    |   movel(p[0.477621, -0.124066, -0.000100, 0.000000, -3.141593, 0.000000],accel_mss,speed_ms,0,0.000)
    |   movel(p[0.477798, -0.124158, -0.000100, 0.000000, -3.141593, 0.000000],accel_mss,speed_ms,0,0.000)
    |   movel(p[0.478109, -0.124225, -0.000100, 0.000000, -3.141593, 0.000000],accel_mss,speed_ms,0,0.000)
    |   movel(p[0.479198, -0.124264, -0.000100, 0.000000, -3.141593, 0.000000],accel_mss,speed_ms,0,blend_radius_m)
    |   movel(p[0.480587, -0.124288, -0.000100, 0.000000, -3.141593, 0.000000],accel_mss,speed_ms,0,blend_radius_m)
    |   movel(p[0.482336, -0.124287, -0.000100, 0.000000, -3.141593, 0.000000],accel_mss,speed_ms,0,blend_radius_m)
    |   movel(p[0.485028, -0.124276, -0.000100, 0.000000, -3.141593, 0.000000],accel_mss,speed_ms,0,blend_radius_m)
    |   movel(p[0.485945, -0.124305, -0.000100, 0.000000, -3.141593, 0.000000],accel_mss,speed_ms,0,blend_radius_m)
    |   movel(p[0.486397, -0.124386, -0.000100, 0.000000, -3.141593, 0.000000],accel_mss,speed_ms,0,0.000)
    |   movel(p[0.486582, -0.124567, -0.000100, 0.000000, -3.141593, 0.000000],accel_mss,speed_ms,0,0.000)
    |   speed_ms    = 0.050
    |   movel(p[0.486582, -0.124567, 0.003000, 0.000000, -3.141593, 0.000000],accel_mss,speed_ms,0,blend_radius_m)
    |   speed_ms    = 1.000
    |   movel(p[0.486582, -0.124567, 0.015000, 0.000000, -3.141593, 0.000000],accel_mss,speed_ms,0,blend_radius_m)
    |   movel(p[0.485986, -0.113553, 0.015000, 0.000000, -3.141593, 0.000000],accel_mss,speed_ms,0,blend_radius_m)
    |   movel(p[0.485986, -0.113553, 0.003000, 0.000000, -3.141593, 0.000000],accel_mss,speed_ms,0,blend_radius_m)
    |   speed_ms    = 0.050
    |   movel(p[0.485986, -0.113553, -0.000100, 0.000000, -3.141593, 0.000000],accel_mss,speed_ms,0,blend_radius_m)
    |   speed_ms    = 0.083
    |   movel(p[0.483901, -0.113573, -0.000100, 0.000000, -3.141593, 0.000000],accel_mss,speed_ms,0,blend_radius_m)
    |   movel(p[0.481817, -0.113593, -0.000100, 0.000000, -3.141593, 0.000000],accel_mss,speed_ms,0,blend_radius_m)
    |   movel(p[0.479732, -0.113613, -0.000100, 0.000000, -3.141593, 0.000000],accel_mss,speed_ms,0,blend_radius_m)
    |   movel(p[0.477648, -0.113633, -0.000100, 0.000000, -3.141593, 0.000000],accel_mss,speed_ms,0,blend_radius_m)
    |   movel(p[0.477670, -0.113088, -0.000100, 0.000000, -3.141593, 0.000000],accel_mss,speed_ms,0,blend_radius_m)
    |   movel(p[0.477692, -0.112543, -0.000100, 0.000000, -3.141593, 0.000000],accel_mss,speed_ms,0,blend_radius_m)
    |   movel(p[0.477714, -0.111998, -0.000100, 0.000000, -3.141593, 0.000000],accel_mss,speed_ms,0,blend_radius_m)
    |   movel(p[0.477736, -0.111453, -0.000100, 0.000000, -3.141593, 0.000000],accel_mss,speed_ms,0,blend_radius_m)
    |   movel(p[0.478467, -0.111432, -0.000100, 0.000000, -3.141593, 0.000000],accel_mss,speed_ms,0,blend_radius_m)
    |   movel(p[0.479198, -0.111410, -0.000100, 0.000000, -3.141593, 0.000000],accel_mss,speed_ms,0,blend_radius_m)
    |   movel(p[0.479930, -0.111389, -0.000100, 0.000000, -3.141593, 0.000000],accel_mss,speed_ms,0,blend_radius_m)
    |   movel(p[0.480661, -0.111367, -0.000100, 0.000000, -3.141593, 0.000000],accel_mss,speed_ms,0,blend_radius_m)
    |   movel(p[0.480661, -0.110676, -0.000100, 0.000000, -3.141593, 0.000000],accel_mss,speed_ms,0,blend_radius_m)
    |   movel(p[0.480660, -0.109985, -0.000100, 0.000000, -3.141593, 0.000000],accel_mss,speed_ms,0,blend_radius_m)
    |   movel(p[0.480609, -0.108937, -0.000100, 0.000000, -3.141593, 0.000000],accel_mss,speed_ms,0,blend_radius_m)
    |   movel(p[0.480436, -0.108259, -0.000100, 0.000000, -3.141593, 0.000000],accel_mss,speed_ms,0,blend_radius_m)
    |   movel(p[0.480104, -0.107790, -0.000100, 0.000000, -3.141593, 0.000000],accel_mss,speed_ms,0,blend_radius_m)
    |   movel(p[0.479569, -0.107429, -0.000100, 0.000000, -3.141593, 0.000000],accel_mss,speed_ms,0,blend_radius_m)
    |   movel(p[0.478777, -0.107208, -0.000100, 0.000000, -3.141593, 0.000000],accel_mss,speed_ms,0,blend_radius_m)
    |   movel(p[0.477995, -0.107283, -0.000100, 0.000000, -3.141593, 0.000000],accel_mss,speed_ms,0,blend_radius_m)
    |   movel(p[0.477300, -0.107648, -0.000100, 0.000000, -3.141593, 0.000000],accel_mss,speed_ms,0,blend_radius_m)
    |   movel(p[0.476760, -0.108264, -0.000100, 0.000000, -3.141593, 0.000000],accel_mss,speed_ms,0,blend_radius_m)
    |   movel(p[0.476590, -0.108694, -0.000100, 0.000000, -3.141593, 0.000000],accel_mss,speed_ms,0,0.000)
    |   movel(p[0.476506, -0.109313, -0.000100, 0.000000, -3.141593, 0.000000],accel_mss,speed_ms,0,blend_radius_m)
    |   movel(p[0.476469, -0.110393, -0.000100, 0.000000, -3.141593, 0.000000],accel_mss,speed_ms,0,blend_radius_m)
    |   movel(p[0.476462, -0.112991, -0.000100, 0.000000, -3.141593, 0.000000],accel_mss,speed_ms,0,blend_radius_m)
    |   movel(p[0.476452, -0.114733, -0.000100, 0.000000, -3.141593, 0.000000],accel_mss,speed_ms,0,blend_radius_m)
    |   movel(p[0.476422, -0.116072, -0.000100, 0.000000, -3.141593, 0.000000],accel_mss,speed_ms,0,blend_radius_m)
    |   movel(p[0.476382, -0.117168, -0.000100, 0.000000, -3.141593, 0.000000],accel_mss,speed_ms,0,blend_radius_m)
    |   movel(p[0.476227, -0.117255, -0.000100, 0.000000, -3.141593, 0.000000],accel_mss,speed_ms,0,0.000)
    |   movel(p[0.475927, -0.117449, -0.000100, 0.000000, -3.141593, 0.000000],accel_mss,speed_ms,0,0.000)
    |   movel(p[0.475575, -0.117691, -0.000100, 0.000000, -3.141593, 0.000000],accel_mss,speed_ms,0,0.000)
    |   movel(p[0.475185, -0.117979, -0.000100, 0.000000, -3.141593, 0.000000],accel_mss,speed_ms,0,0.000)
    |   movel(p[0.474689, -0.118354, -0.000100, 0.000000, -3.141593, 0.000000],accel_mss,speed_ms,0,blend_radius_m)
    |   movel(p[0.474193, -0.118730, -0.000100, 0.000000, -3.141593, 0.000000],accel_mss,speed_ms,0,blend_radius_m)
    |   movel(p[0.474216, -0.116123, -0.000100, 0.000000, -3.141593, 0.000000],accel_mss,speed_ms,0,blend_radius_m)
    |   movel(p[0.474240, -0.113517, -0.000100, 0.000000, -3.141593, 0.000000],accel_mss,speed_ms,0,blend_radius_m)
    |   movel(p[0.474276, -0.110264, -0.000100, 0.000000, -3.141593, 0.000000],accel_mss,speed_ms,0,blend_radius_m)
    |   movel(p[0.474325, -0.108952, -0.000100, 0.000000, -3.141593, 0.000000],accel_mss,speed_ms,0,blend_radius_m)
    |   movel(p[0.474421, -0.108190, -0.000100, 0.000000, -3.141593, 0.000000],accel_mss,speed_ms,0,blend_radius_m)
    |   movel(p[0.474607, -0.107610, -0.000100, 0.000000, -3.141593, 0.000000],accel_mss,speed_ms,0,blend_radius_m)
    |   movel(p[0.475305, -0.106500, -0.000100, 0.000000, -3.141593, 0.000000],accel_mss,speed_ms,0,blend_radius_m)
    |   movel(p[0.476224, -0.105682, -0.000100, 0.000000, -3.141593, 0.000000],accel_mss,speed_ms,0,blend_radius_m)
    |   movel(p[0.477346, -0.105184, -0.000100, 0.000000, -3.141593, 0.000000],accel_mss,speed_ms,0,blend_radius_m)
    |   movel(p[0.478636, -0.105013, -0.000100, 0.000000, -3.141593, 0.000000],accel_mss,speed_ms,0,blend_radius_m)
    |   movel(p[0.479885, -0.105172, -0.000100, 0.000000, -3.141593, 0.000000],accel_mss,speed_ms,0,blend_radius_m)
    |   movel(p[0.480979, -0.105640, -0.000100, 0.000000, -3.141593, 0.000000],accel_mss,speed_ms,0,blend_radius_m)
    |   movel(p[0.481876, -0.106408, -0.000100, 0.000000, -3.141593, 0.000000],accel_mss,speed_ms,0,blend_radius_m)
    |   movel(p[0.482547, -0.107441, -0.000100, 0.000000, -3.141593, 0.000000],accel_mss,speed_ms,0,blend_radius_m)
    |   movel(p[0.482753, -0.107943, -0.000100, 0.000000, -3.141593, 0.000000],accel_mss,speed_ms,0,blend_radius_m)
    |   movel(p[0.482884, -0.108421, -0.000100, 0.000000, -3.141593, 0.000000],accel_mss,speed_ms,0,0.000)
    |   movel(p[0.482966, -0.108996, -0.000100, 0.000000, -3.141593, 0.000000],accel_mss,speed_ms,0,blend_radius_m)
    |   movel(p[0.483025, -0.109826, -0.000100, 0.000000, -3.141593, 0.000000],accel_mss,speed_ms,0,blend_radius_m)
    |   movel(p[0.483064, -0.110597, -0.000100, 0.000000, -3.141593, 0.000000],accel_mss,speed_ms,0,blend_radius_m)
    |   movel(p[0.483104, -0.111368, -0.000100, 0.000000, -3.141593, 0.000000],accel_mss,speed_ms,0,blend_radius_m)
    |   movel(p[0.483824, -0.111389, -0.000100, 0.000000, -3.141593, 0.000000],accel_mss,speed_ms,0,blend_radius_m)
    |   movel(p[0.484545, -0.111411, -0.000100, 0.000000, -3.141593, 0.000000],accel_mss,speed_ms,0,blend_radius_m)
    |   movel(p[0.485265, -0.111432, -0.000100, 0.000000, -3.141593, 0.000000],accel_mss,speed_ms,0,blend_radius_m)
    |   movel(p[0.485986, -0.111453, -0.000100, 0.000000, -3.141593, 0.000000],accel_mss,speed_ms,0,blend_radius_m)
    |   movel(p[0.485986, -0.111978, -0.000100, 0.000000, -3.141593, 0.000000],accel_mss,speed_ms,0,blend_radius_m)
    |   movel(p[0.485986, -0.112503, -0.000100, 0.000000, -3.141593, 0.000000],accel_mss,speed_ms,0,blend_radius_m)
    |   movel(p[0.485986, -0.113028, -0.000100, 0.000000, -3.141593, 0.000000],accel_mss,speed_ms,0,blend_radius_m)
    |   movel(p[0.485986, -0.113553, -0.000100, 0.000000, -3.141593, 0.000000],accel_mss,speed_ms,0,blend_radius_m)
    |   speed_ms    = 0.050
    |   movel(p[0.485986, -0.113553, 0.003000, 0.000000, -3.141593, 0.000000],accel_mss,speed_ms,0,blend_radius_m)
    |   speed_ms    = 1.000
    |   movel(p[0.485986, -0.113553, 0.015000, 0.000000, -3.141593, 0.000000],accel_mss,speed_ms,0,blend_radius_m)
    |   movel(p[0.487186, -0.112578, 0.015000, 0.000000, -3.141593, 0.000000],accel_mss,speed_ms,0,blend_radius_m)
    |   movel(p[0.487186, -0.112578, 0.003000, 0.000000, -3.141593, 0.000000],accel_mss,speed_ms,0,blend_radius_m)
    |   speed_ms    = 0.050
    |   movel(p[0.487186, -0.112578, -0.000100, 0.000000, -3.141593, 0.000000],accel_mss,speed_ms,0,blend_radius_m)
    |   speed_ms    = 0.083
    |   movel(p[0.487186, -0.110516, -0.000100, 0.000000, -3.141593, 0.000000],accel_mss,speed_ms,0,blend_radius_m)
    |   movel(p[0.487186, -0.108453, -0.000100, 0.000000, -3.141593, 0.000000],accel_mss,speed_ms,0,blend_radius_m)
    |   movel(p[0.487730, -0.108431, -0.000100, 0.000000, -3.141593, 0.000000],accel_mss,speed_ms,0,blend_radius_m)
    |   movel(p[0.488273, -0.108409, -0.000100, 0.000000, -3.141593, 0.000000],accel_mss,speed_ms,0,blend_radius_m)
    |   movel(p[0.488817, -0.108387, -0.000100, 0.000000, -3.141593, 0.000000],accel_mss,speed_ms,0,blend_radius_m)
    |   movel(p[0.489361, -0.108365, -0.000100, 0.000000, -3.141593, 0.000000],accel_mss,speed_ms,0,blend_radius_m)
    |   movel(p[0.489361, -0.109118, -0.000100, 0.000000, -3.141593, 0.000000],accel_mss,speed_ms,0,blend_radius_m)
    |   movel(p[0.489361, -0.109872, -0.000100, 0.000000, -3.141593, 0.000000],accel_mss,speed_ms,0,blend_radius_m)
    |   movel(p[0.489361, -0.110625, -0.000100, 0.000000, -3.141593, 0.000000],accel_mss,speed_ms,0,blend_radius_m)
    |   movel(p[0.489361, -0.111378, -0.000100, 0.000000, -3.141593, 0.000000],accel_mss,speed_ms,0,blend_radius_m)
    |   movel(p[0.490055, -0.111378, -0.000100, 0.000000, -3.141593, 0.000000],accel_mss,speed_ms,0,blend_radius_m)
    |   movel(p[0.490748, -0.111378, -0.000100, 0.000000, -3.141593, 0.000000],accel_mss,speed_ms,0,blend_radius_m)
    |   movel(p[0.491480, -0.111365, -0.000100, 0.000000, -3.141593, 0.000000],accel_mss,speed_ms,0,blend_radius_m)
    |   movel(p[0.491955, -0.111319, -0.000100, 0.000000, -3.141593, 0.000000],accel_mss,speed_ms,0,0.000)
    |   movel(p[0.492306, -0.111231, -0.000100, 0.000000, -3.141593, 0.000000],accel_mss,speed_ms,0,0.000)
    |   movel(p[0.492616, -0.111084, -0.000100, 0.000000, -3.141593, 0.000000],accel_mss,speed_ms,0,0.000)
    |   movel(p[0.493345, -0.110305, -0.000100, 0.000000, -3.141593, 0.000000],accel_mss,speed_ms,0,blend_radius_m)
    |   movel(p[0.493590, -0.109242, -0.000100, 0.000000, -3.141593, 0.000000],accel_mss,speed_ms,0,blend_radius_m)
    |   movel(p[0.493285, -0.108194, -0.000100, 0.000000, -3.141593, 0.000000],accel_mss,speed_ms,0,blend_radius_m)
    |   movel(p[0.492513, -0.107458, -0.000100, 0.000000, -3.141593, 0.000000],accel_mss,speed_ms,0,blend_radius_m)
    |   movel(p[0.492066, -0.107302, -0.000100, 0.000000, -3.141593, 0.000000],accel_mss,speed_ms,0,0.000)
    |   movel(p[0.491411, -0.107223, -0.000100, 0.000000, -3.141593, 0.000000],accel_mss,speed_ms,0,blend_radius_m)
    |   movel(p[0.490300, -0.107186, -0.000100, 0.000000, -3.141593, 0.000000],accel_mss,speed_ms,0,blend_radius_m)
    |   movel(p[0.487851, -0.107178, -0.000100, 0.000000, -3.141593, 0.000000],accel_mss,speed_ms,0,blend_radius_m)
    |   movel(p[0.485781, -0.107178, -0.000100, 0.000000, -3.141593, 0.000000],accel_mss,speed_ms,0,blend_radius_m)
    |   movel(p[0.483711, -0.107178, -0.000100, 0.000000, -3.141593, 0.000000],accel_mss,speed_ms,0,blend_radius_m)
    |   movel(p[0.483480, -0.106822, -0.000100, 0.000000, -3.141593, 0.000000],accel_mss,speed_ms,0,0.000)
    |   movel(p[0.483249, -0.106466, -0.000100, 0.000000, -3.141593, 0.000000],accel_mss,speed_ms,0,0.000)
    |   movel(p[0.483043, -0.106166, -0.000100, 0.000000, -3.141593, 0.000000],accel_mss,speed_ms,0,0.000)
    |   movel(p[0.482805, -0.105852, -0.000100, 0.000000, -3.141593, 0.000000],accel_mss,speed_ms,0,0.000)
    |   movel(p[0.482573, -0.105572, -0.000100, 0.000000, -3.141593, 0.000000],accel_mss,speed_ms,0,0.000)
    |   movel(p[0.482387, -0.105378, -0.000100, 0.000000, -3.141593, 0.000000],accel_mss,speed_ms,0,0.000)
    |   movel(p[0.482187, -0.105191, -0.000100, 0.000000, -3.141593, 0.000000],accel_mss,speed_ms,0,0.000)
    |   movel(p[0.481987, -0.105003, -0.000100, 0.000000, -3.141593, 0.000000],accel_mss,speed_ms,0,0.000)
    |   movel(p[0.484482, -0.104984, -0.000100, 0.000000, -3.141593, 0.000000],accel_mss,speed_ms,0,blend_radius_m)
    |   movel(p[0.486978, -0.104964, -0.000100, 0.000000, -3.141593, 0.000000],accel_mss,speed_ms,0,blend_radius_m)
    |   movel(p[0.489633, -0.104952, -0.000100, 0.000000, -3.141593, 0.000000],accel_mss,speed_ms,0,blend_radius_m)
    |   movel(p[0.491149, -0.104975, -0.000100, 0.000000, -3.141593, 0.000000],accel_mss,speed_ms,0,blend_radius_m)
    |   movel(p[0.492126, -0.105033, -0.000100, 0.000000, -3.141593, 0.000000],accel_mss,speed_ms,0,blend_radius_m)
    |   movel(p[0.492740, -0.105148, -0.000100, 0.000000, -3.141593, 0.000000],accel_mss,speed_ms,0,blend_radius_m)
    |   movel(p[0.494613, -0.106288, -0.000100, 0.000000, -3.141593, 0.000000],accel_mss,speed_ms,0,blend_radius_m)
    |   movel(p[0.495680, -0.108227, -0.000100, 0.000000, -3.141593, 0.000000],accel_mss,speed_ms,0,blend_radius_m)
    |   movel(p[0.495658, -0.110448, -0.000100, 0.000000, -3.141593, 0.000000],accel_mss,speed_ms,0,blend_radius_m)
    |   movel(p[0.494549, -0.112360, -0.000100, 0.000000, -3.141593, 0.000000],accel_mss,speed_ms,0,blend_radius_m)
    |   movel(p[0.493823, -0.112964, -0.000100, 0.000000, -3.141593, 0.000000],accel_mss,speed_ms,0,blend_radius_m)
    |   movel(p[0.493066, -0.113356, -0.000100, 0.000000, -3.141593, 0.000000],accel_mss,speed_ms,0,blend_radius_m)
    |   movel(p[0.492132, -0.113595, -0.000100, 0.000000, -3.141593, 0.000000],accel_mss,speed_ms,0,blend_radius_m)
    |   movel(p[0.490829, -0.113732, -0.000100, 0.000000, -3.141593, 0.000000],accel_mss,speed_ms,0,blend_radius_m)
    |   movel(p[0.490100, -0.113777, -0.000100, 0.000000, -3.141593, 0.000000],accel_mss,speed_ms,0,blend_radius_m)
    |   movel(p[0.489371, -0.113823, -0.000100, 0.000000, -3.141593, 0.000000],accel_mss,speed_ms,0,blend_radius_m)
    |   movel(p[0.489350, -0.114543, -0.000100, 0.000000, -3.141593, 0.000000],accel_mss,speed_ms,0,blend_radius_m)
    |   movel(p[0.489329, -0.115263, -0.000100, 0.000000, -3.141593, 0.000000],accel_mss,speed_ms,0,blend_radius_m)
    |   movel(p[0.489307, -0.115983, -0.000100, 0.000000, -3.141593, 0.000000],accel_mss,speed_ms,0,blend_radius_m)
    |   movel(p[0.489286, -0.116703, -0.000100, 0.000000, -3.141593, 0.000000],accel_mss,speed_ms,0,blend_radius_m)
    |   movel(p[0.488761, -0.116703, -0.000100, 0.000000, -3.141593, 0.000000],accel_mss,speed_ms,0,blend_radius_m)
    |   movel(p[0.488236, -0.116703, -0.000100, 0.000000, -3.141593, 0.000000],accel_mss,speed_ms,0,blend_radius_m)
    |   movel(p[0.487711, -0.116703, -0.000100, 0.000000, -3.141593, 0.000000],accel_mss,speed_ms,0,blend_radius_m)
    |   movel(p[0.487186, -0.116703, -0.000100, 0.000000, -3.141593, 0.000000],accel_mss,speed_ms,0,blend_radius_m)
    |   movel(p[0.487186, -0.114641, -0.000100, 0.000000, -3.141593, 0.000000],accel_mss,speed_ms,0,blend_radius_m)
    |   movel(p[0.487186, -0.112578, -0.000100, 0.000000, -3.141593, 0.000000],accel_mss,speed_ms,0,blend_radius_m)
    |   speed_ms    = 0.050
    |   movel(p[0.487186, -0.112578, 0.003000, 0.000000, -3.141593, 0.000000],accel_mss,speed_ms,0,blend_radius_m)
    |   speed_ms    = 1.000
    |   movel(p[0.487186, -0.112578, 0.015000, 0.000000, -3.141593, 0.000000],accel_mss,speed_ms,0,blend_radius_m)
    |   movel(p[0.475139, -0.094856, 0.015000, 0.000000, -3.141593, 0.000000],accel_mss,speed_ms,0,blend_radius_m)
    |   movel(p[0.475139, -0.094856, 0.003000, 0.000000, -3.141593, 0.000000],accel_mss,speed_ms,0,blend_radius_m)
    |   speed_ms    = 0.050
    |   movel(p[0.475139, -0.094856, -0.000100, 0.000000, -3.141593, 0.000000],accel_mss,speed_ms,0,blend_radius_m)
    |   speed_ms    = 0.083
    |   movel(p[0.474976, -0.094899, -0.000100, 0.000000, -3.141593, 0.000000],accel_mss,speed_ms,0,0.000)
    |   movel(p[0.474802, -0.094997, -0.000100, 0.000000, -3.141593, 0.000000],accel_mss,speed_ms,0,0.000)
    |   movel(p[0.474599, -0.095127, -0.000100, 0.000000, -3.141593, 0.000000],accel_mss,speed_ms,0,0.000)
    |   movel(p[0.474386, -0.095281, -0.000100, 0.000000, -3.141593, 0.000000],accel_mss,speed_ms,0,0.000)
    |   movel(p[0.474130, -0.095462, -0.000100, 0.000000, -3.141593, 0.000000],accel_mss,speed_ms,0,0.000)
    |   movel(p[0.473789, -0.095676, -0.000100, 0.000000, -3.141593, 0.000000],accel_mss,speed_ms,0,0.000)
    |   movel(p[0.473427, -0.095886, -0.000100, 0.000000, -3.141593, 0.000000],accel_mss,speed_ms,0,0.000)
    |   movel(p[0.473097, -0.096058, -0.000100, 0.000000, -3.141593, 0.000000],accel_mss,speed_ms,0,0.000)
    |   movel(p[0.472772, -0.096227, -0.000100, 0.000000, -3.141593, 0.000000],accel_mss,speed_ms,0,0.000)
    |   movel(p[0.472423, -0.096425, -0.000100, 0.000000, -3.141593, 0.000000],accel_mss,speed_ms,0,0.000)
    |   movel(p[0.472103, -0.096621, -0.000100, 0.000000, -3.141593, 0.000000],accel_mss,speed_ms,0,0.000)
    |   movel(p[0.471872, -0.096781, -0.000100, 0.000000, -3.141593, 0.000000],accel_mss,speed_ms,0,0.000)
    |   movel(p[0.471685, -0.096914, -0.000100, 0.000000, -3.141593, 0.000000],accel_mss,speed_ms,0,0.000)
    |   movel(p[0.471508, -0.097026, -0.000100, 0.000000, -3.141593, 0.000000],accel_mss,speed_ms,0,0.000)
    |   movel(p[0.471356, -0.097111, -0.000100, 0.000000, -3.141593, 0.000000],accel_mss,speed_ms,0,0.000)
    |   movel(p[0.471201, -0.097144, -0.000100, 0.000000, -3.141593, 0.000000],accel_mss,speed_ms,0,0.000)
    |   movel(p[0.470928, -0.097257, -0.000100, 0.000000, -3.141593, 0.000000],accel_mss,speed_ms,0,0.000)
    |   movel(p[0.470606, -0.097398, -0.000100, 0.000000, -3.141593, 0.000000],accel_mss,speed_ms,0,0.000)
    |   movel(p[0.470248, -0.097565, -0.000100, 0.000000, -3.141593, 0.000000],accel_mss,speed_ms,0,0.000)
    |   movel(p[0.468933, -0.098159, -0.000100, 0.000000, -3.141593, 0.000000],accel_mss,speed_ms,0,blend_radius_m)
    |   movel(p[0.467453, -0.098761, -0.000100, 0.000000, -3.141593, 0.000000],accel_mss,speed_ms,0,blend_radius_m)
    |   movel(p[0.466092, -0.099268, -0.000100, 0.000000, -3.141593, 0.000000],accel_mss,speed_ms,0,blend_radius_m)
    |   movel(p[0.465361, -0.099462, -0.000100, 0.000000, -3.141593, 0.000000],accel_mss,speed_ms,0,blend_radius_m)
    |   movel(p[0.465128, -0.099511, -0.000100, 0.000000, 3.141593, 0.000000],accel_mss,speed_ms,0,0.000)
    |   movel(p[0.464589, -0.099642, -0.000100, 0.000000, -3.141593, 0.000000],accel_mss,speed_ms,0,blend_radius_m)
    |   movel(p[0.463949, -0.099802, -0.000100, 0.000000, -3.141593, 0.000000],accel_mss,speed_ms,0,blend_radius_m)
    |   movel(p[0.463261, -0.099980, -0.000100, 0.000000, -3.141593, 0.000000],accel_mss,speed_ms,0,blend_radius_m)
    |   movel(p[0.461204, -0.100416, -0.000100, 0.000000, -3.141593, 0.000000],accel_mss,speed_ms,0,blend_radius_m)
    |   movel(p[0.458958, -0.100699, -0.000100, 0.000000, -3.141593, 0.000000],accel_mss,speed_ms,0,blend_radius_m)
    |   movel(p[0.456502, -0.100831, -0.000100, 0.000000, -3.141593, 0.000000],accel_mss,speed_ms,0,blend_radius_m)
    |   movel(p[0.453811, -0.100812, -0.000100, 0.000000, -3.141593, 0.000000],accel_mss,speed_ms,0,blend_radius_m)
    |   movel(p[0.451778, -0.100741, -0.000100, 0.000000, -3.141593, 0.000000],accel_mss,speed_ms,0,blend_radius_m)
    |   movel(p[0.450704, -0.100686, -0.000100, 0.000000, -3.141593, 0.000000],accel_mss,speed_ms,0,blend_radius_m)
    |   movel(p[0.449901, -0.100617, -0.000100, 0.000000, -3.141593, 0.000000],accel_mss,speed_ms,0,blend_radius_m)
    |   movel(p[0.449023, -0.100506, -0.000100, 0.000000, -3.141593, 0.000000],accel_mss,speed_ms,0,blend_radius_m)
    |   movel(p[0.448418, -0.100401, -0.000100, 0.000000, -3.141593, 0.000000],accel_mss,speed_ms,0,blend_radius_m)
    |   movel(p[0.447790, -0.100254, -0.000100, 0.000000, -3.141593, 0.000000],accel_mss,speed_ms,0,blend_radius_m)
    |   movel(p[0.447240, -0.100096, -0.000100, 0.000000, -3.141593, 0.000000],accel_mss,speed_ms,0,blend_radius_m)
    |   movel(p[0.446986, -0.099972, -0.000100, 0.000000, -3.141593, 0.000000],accel_mss,speed_ms,0,0.000)
    |   movel(p[0.446886, -0.099918, -0.000100, 0.000000, -3.141593, 0.000000],accel_mss,speed_ms,0,0.000)
    |   movel(p[0.446638, -0.099819, -0.000100, 0.000000, -3.141593, 0.000000],accel_mss,speed_ms,0,0.000)
    |   movel(p[0.446338, -0.099710, -0.000100, 0.000000, -3.141593, 0.000000],accel_mss,speed_ms,0,0.000)
    |   movel(p[0.446011, -0.099599, -0.000100, 0.000000, 3.141593, 0.000000],accel_mss,speed_ms,0,0.000)
    |   movel(p[0.445321, -0.099341, -0.000100, 0.000000, -3.141593, 0.000000],accel_mss,speed_ms,0,blend_radius_m)
    |   movel(p[0.444524, -0.098979, -0.000100, 0.000000, -3.141593, 0.000000],accel_mss,speed_ms,0,blend_radius_m)
    |   movel(p[0.443794, -0.098604, -0.000100, 0.000000, -3.141593, 0.000000],accel_mss,speed_ms,0,blend_radius_m)
    |   movel(p[0.443383, -0.098326, -0.000100, 0.000000, -3.141593, 0.000000],accel_mss,speed_ms,0,0.000)
    |   movel(p[0.443297, -0.098263, -0.000100, 0.000000, -3.141593, 0.000000],accel_mss,speed_ms,0,0.000)
    |   movel(p[0.443181, -0.098227, -0.000100, 0.000000, -3.141593, 0.000000],accel_mss,speed_ms,0,0.000)
    |   movel(p[0.442974, -0.098181, -0.000100, 0.000000, -3.141593, 0.000000],accel_mss,speed_ms,0,0.000)
    |   movel(p[0.442768, -0.098040, -0.000100, 0.000000, -3.141593, 0.000000],accel_mss,speed_ms,0,0.000)
    |   movel(p[0.442523, -0.097850, -0.000100, 0.000000, -3.141593, 0.000000],accel_mss,speed_ms,0,0.000)
    |   movel(p[0.442241, -0.097636, -0.000100, 0.000000, -3.141593, 0.000000],accel_mss,speed_ms,0,0.000)
    |   movel(p[0.441918, -0.097415, -0.000100, 0.000000, -3.141593, 0.000000],accel_mss,speed_ms,0,0.000)
    |   movel(p[0.441606, -0.097222, -0.000100, 0.000000, -3.141593, 0.000000],accel_mss,speed_ms,0,0.000)
    |   movel(p[0.441359, -0.097092, -0.000100, 0.000000, -3.141593, 0.000000],accel_mss,speed_ms,0,0.000)
    |   movel(p[0.441130, -0.096970, -0.000100, 0.000000, -3.141593, 0.000000],accel_mss,speed_ms,0,0.000)
    |   movel(p[0.440880, -0.096806, -0.000100, 0.000000, -3.141593, 0.000000],accel_mss,speed_ms,0,0.000)
    |   movel(p[0.440646, -0.096628, -0.000100, 0.000000, -3.141593, 0.000000],accel_mss,speed_ms,0,0.000)
    |   movel(p[0.440470, -0.096463, -0.000100, 0.000000, -3.141593, 0.000000],accel_mss,speed_ms,0,0.000)
    |   movel(p[0.440318, -0.096316, -0.000100, 0.000000, -3.141593, 0.000000],accel_mss,speed_ms,0,0.000)
    |   movel(p[0.440160, -0.096191, -0.000100, 0.000000, -3.141593, 0.000000],accel_mss,speed_ms,0,0.000)
    |   movel(p[0.440017, -0.096103, -0.000100, 0.000000, -3.141593, 0.000000],accel_mss,speed_ms,0,0.000)
    |   movel(p[0.439640, -0.095963, -0.000100, 0.000000, -3.141593, 0.000000],accel_mss,speed_ms,0,0.000)
    |   movel(p[0.437918, -0.094263, -0.000100, 0.000000, -3.141593, 0.000000],accel_mss,speed_ms,0,blend_radius_m)
    |   movel(p[0.436284, -0.092619, -0.000100, 0.000000, -3.141593, 0.000000],accel_mss,speed_ms,0,blend_radius_m)
    |   movel(p[0.435945, -0.092125, -0.000100, 0.000000, -3.141593, 0.000000],accel_mss,speed_ms,0,blend_radius_m)
    |   movel(p[0.435776, -0.091780, -0.000100, 0.000000, -3.141593, 0.000000],accel_mss,speed_ms,0,0.000)
    |   movel(p[0.435584, -0.091437, -0.000100, 0.000000, -3.141593, 0.000000],accel_mss,speed_ms,0,0.000)
    |   movel(p[0.435386, -0.091123, -0.000100, 0.000000, -3.141593, 0.000000],accel_mss,speed_ms,0,0.000)
    |   movel(p[0.435198, -0.090867, -0.000100, 0.000000, -3.141593, 0.000000],accel_mss,speed_ms,0,0.000)
    |   movel(p[0.434504, -0.089799, -0.000100, 0.000000, -3.141593, 0.000000],accel_mss,speed_ms,0,blend_radius_m)
    |   movel(p[0.433763, -0.088207, -0.000100, 0.000000, -3.141593, 0.000000],accel_mss,speed_ms,0,blend_radius_m)
    |   movel(p[0.433087, -0.086395, -0.000100, 0.000000, -3.141593, 0.000000],accel_mss,speed_ms,0,blend_radius_m)
    |   movel(p[0.432581, -0.084603, -0.000100, 0.000000, -3.141593, 0.000000],accel_mss,speed_ms,0,blend_radius_m)
    |   movel(p[0.432399, -0.083394, -0.000100, 0.000000, -3.141593, 0.000000],accel_mss,speed_ms,0,blend_radius_m)
    |   movel(p[0.432295, -0.081278, -0.000100, 0.000000, -3.141593, 0.000000],accel_mss,speed_ms,0,blend_radius_m)
    |   movel(p[0.432239, -0.079022, -0.000100, 0.000000, -3.141593, 0.000000],accel_mss,speed_ms,0,blend_radius_m)
    |   movel(p[0.432399, -0.078730, -0.000100, 0.000000, -3.141593, 0.000000],accel_mss,speed_ms,0,0.000)
    |   movel(p[0.432705, -0.078872, -0.000100, 0.000000, -3.141593, 0.000000],accel_mss,speed_ms,0,0.000)
    |   movel(p[0.432963, -0.079076, -0.000100, 0.000000, 3.141593, 0.000000],accel_mss,speed_ms,0,0.000)
    |   movel(p[0.433243, -0.079336, -0.000100, 0.000000, -3.141593, 0.000000],accel_mss,speed_ms,0,0.000)
    |   movel(p[0.433523, -0.079601, -0.000100, 0.000000, -3.141593, 0.000000],accel_mss,speed_ms,0,0.000)
    |   movel(p[0.433784, -0.079825, -0.000100, 0.000000, -3.141593, 0.000000],accel_mss,speed_ms,0,0.000)
    |   movel(p[0.434008, -0.079998, -0.000100, 0.000000, 3.141593, 0.000000],accel_mss,speed_ms,0,0.000)
    |   movel(p[0.434186, -0.080057, -0.000100, 0.000000, -3.141593, 0.000000],accel_mss,speed_ms,0,0.000)
    |   movel(p[0.434378, -0.080205, -0.000100, 0.000000, -3.141593, 0.000000],accel_mss,speed_ms,0,0.000)
    |   movel(p[0.434600, -0.080399, -0.000100, 0.000000, -3.141593, 0.000000],accel_mss,speed_ms,0,0.000)
    |   movel(p[0.434836, -0.080628, -0.000100, 0.000000, -3.141593, 0.000000],accel_mss,speed_ms,0,0.000)
    |   movel(p[0.435070, -0.080858, -0.000100, 0.000000, -3.141593, 0.000000],accel_mss,speed_ms,0,0.000)
    |   movel(p[0.435289, -0.081052, -0.000100, 0.000000, -3.141593, 0.000000],accel_mss,speed_ms,0,0.000)
    |   movel(p[0.435477, -0.081202, -0.000100, 0.000000, -3.141593, 0.000000],accel_mss,speed_ms,0,0.000)
    |   movel(p[0.435638, -0.081254, -0.000100, 0.000000, -3.141593, 0.000000],accel_mss,speed_ms,0,0.000)
    |   movel(p[0.435881, -0.081427, -0.000100, 0.000000, -3.141593, 0.000000],accel_mss,speed_ms,0,0.000)
    |   movel(p[0.436166, -0.081645, -0.000100, 0.000000, -3.141593, 0.000000],accel_mss,speed_ms,0,0.000)
    |   movel(p[0.436478, -0.081903, -0.000100, 0.000000, -3.141593, 0.000000],accel_mss,speed_ms,0,0.000)
    |   movel(p[0.436792, -0.082162, -0.000100, 0.000000, -3.141593, 0.000000],accel_mss,speed_ms,0,0.000)
    |   movel(p[0.437080, -0.082380, -0.000100, 0.000000, -3.141593, 0.000000],accel_mss,speed_ms,0,0.000)
    |   movel(p[0.437325, -0.082551, -0.000100, 0.000000, -3.141593, 0.000000],accel_mss,speed_ms,0,0.000)
    |   movel(p[0.437491, -0.082597, -0.000100, 0.000000, -3.141593, 0.000000],accel_mss,speed_ms,0,0.000)
    |   movel(p[0.437601, -0.082666, -0.000100, 0.000000, -3.141593, 0.000000],accel_mss,speed_ms,0,0.000)
    |   movel(p[0.437721, -0.082764, -0.000100, 0.000000, -3.141593, 0.000000],accel_mss,speed_ms,0,0.000)
    |   movel(p[0.437836, -0.082878, -0.000100, 0.000000, -3.141593, 0.000000],accel_mss,speed_ms,0,0.000)
    |   movel(p[0.437953, -0.082993, -0.000100, 0.000000, -3.141593, 0.000000],accel_mss,speed_ms,0,0.000)
    |   movel(p[0.438080, -0.083090, -0.000100, 0.000000, -3.141593, 0.000000],accel_mss,speed_ms,0,0.000)
    |   movel(p[0.438199, -0.083158, -0.000100, 0.000000, -3.141593, 0.000000],accel_mss,speed_ms,0,0.000)
    |   movel(p[0.438373, -0.083198, -0.000100, 0.000000, -3.141593, 0.000000],accel_mss,speed_ms,0,0.000)
    |   movel(p[0.438492, -0.083267, -0.000100, 0.000000, -3.141593, 0.000000],accel_mss,speed_ms,0,0.000)
    |   movel(p[0.438619, -0.083364, -0.000100, 0.000000, -3.141593, 0.000000],accel_mss,speed_ms,0,0.000)
    |   movel(p[0.438737, -0.083479, -0.000100, 0.000000, -3.141593, 0.000000],accel_mss,speed_ms,0,0.000)
    |   movel(p[0.438846, -0.083590, -0.000100, 0.000000, -3.141593, 0.000000],accel_mss,speed_ms,0,0.000)
    |   movel(p[0.438950, -0.083671, -0.000100, 0.000000, -3.141593, 0.000000],accel_mss,speed_ms,0,0.000)
    |   movel(p[0.439079, -0.083710, -0.000100, 0.000000, -3.141593, 0.000000],accel_mss,speed_ms,0,0.000)
    |   movel(p[0.439310, -0.083808, -0.000100, 0.000000, -3.141593, 0.000000],accel_mss,speed_ms,0,0.000)
    |   movel(p[0.439526, -0.083954, -0.000100, 0.000000, -3.141593, 0.000000],accel_mss,speed_ms,0,0.000)
    |   movel(p[0.439768, -0.084141, -0.000100, 0.000000, -3.141593, 0.000000],accel_mss,speed_ms,0,0.000)
    |   movel(p[0.440032, -0.084341, -0.000100, 0.000000, 3.141593, 0.000000],accel_mss,speed_ms,0,0.000)
    |   movel(p[0.440315, -0.084527, -0.000100, 0.000000, -3.141593, 0.000000],accel_mss,speed_ms,0,0.000)
    |   movel(p[0.440575, -0.084677, -0.000100, 0.000000, -3.141593, 0.000000],accel_mss,speed_ms,0,0.000)
    |   movel(p[0.440761, -0.084753, -0.000100, 0.000000, -3.141593, 0.000000],accel_mss,speed_ms,0,0.000)
    |   movel(p[0.440921, -0.084809, -0.000100, 0.000000, -3.141593, 0.000000],accel_mss,speed_ms,0,0.000)
    |   movel(p[0.441092, -0.084887, -0.000100, 0.000000, -3.141593, 0.000000],accel_mss,speed_ms,0,0.000)
    |   movel(p[0.441248, -0.084972, -0.000100, 0.000000, -3.141593, 0.000000],accel_mss,speed_ms,0,0.000)
    |   movel(p[0.441361, -0.085053, -0.000100, 0.000000, -3.141593, 0.000000],accel_mss,speed_ms,0,0.000)
    |   movel(p[0.441738, -0.085300, -0.000100, 0.000000, -3.141593, 0.000000],accel_mss,speed_ms,0,0.000)
    |   movel(p[0.443284, -0.086059, -0.000100, 0.000000, -3.141593, 0.000000],accel_mss,speed_ms,0,blend_radius_m)
    |   movel(p[0.444784, -0.086773, -0.000100, 0.000000, -3.141593, 0.000000],accel_mss,speed_ms,0,blend_radius_m)
    |   movel(p[0.445636, -0.087129, -0.000100, 0.000000, -3.141593, 0.000000],accel_mss,speed_ms,0,blend_radius_m)
    |   movel(p[0.445938, -0.087242, -0.000100, 0.000000, -3.141593, 0.000000],accel_mss,speed_ms,0,0.000)
    |   movel(p[0.446368, -0.087404, -0.000100, 0.000000, -3.141593, 0.000000],accel_mss,speed_ms,0,0.000)
    |   movel(p[0.446840, -0.087583, -0.000100, 0.000000, -3.141593, 0.000000],accel_mss,speed_ms,0,blend_radius_m)
    |   movel(p[0.447286, -0.087752, -0.000100, 0.000000, 3.141593, 0.000000],accel_mss,speed_ms,0,0.000)
    |   movel(p[0.447715, -0.087909, -0.000100, 0.000000, -3.141593, 0.000000],accel_mss,speed_ms,0,0.000)
    |   movel(p[0.448138, -0.088051, -0.000100, 0.000000, -3.141593, 0.000000],accel_mss,speed_ms,0,0.000)
    |   movel(p[0.448503, -0.088163, -0.000100, 0.000000, -3.141593, 0.000000],accel_mss,speed_ms,0,0.000)
    |   movel(p[0.448711, -0.088210, -0.000100, 0.000000, -3.141593, 0.000000],accel_mss,speed_ms,0,0.000)
    |   movel(p[0.448946, -0.088252, -0.000100, 0.000000, -3.141593, 0.000000],accel_mss,speed_ms,0,0.000)
    |   movel(p[0.449505, -0.088367, -0.000100, 0.000000, -3.141593, 0.000000],accel_mss,speed_ms,0,blend_radius_m)
    |   movel(p[0.450169, -0.088506, -0.000100, 0.000000, -3.141593, 0.000000],accel_mss,speed_ms,0,blend_radius_m)
    |   movel(p[0.450886, -0.088661, -0.000100, 0.000000, -3.141593, 0.000000],accel_mss,speed_ms,0,blend_radius_m)
    |   movel(p[0.452676, -0.088950, -0.000100, 0.000000, -3.141593, 0.000000],accel_mss,speed_ms,0,blend_radius_m)
    |   movel(p[0.454635, -0.089077, -0.000100, 0.000000, -3.141593, 0.000000],accel_mss,speed_ms,0,blend_radius_m)
    |   movel(p[0.456523, -0.089036, -0.000100, 0.000000, -3.141593, 0.000000],accel_mss,speed_ms,0,blend_radius_m)
    |   movel(p[0.458086, -0.088818, -0.000100, 0.000000, 3.141593, 0.000000],accel_mss,speed_ms,0,blend_radius_m)
    |   movel(p[0.460163, -0.088275, -0.000100, 0.000000, -3.141593, 0.000000],accel_mss,speed_ms,0,blend_radius_m)
    |   movel(p[0.462177, -0.087556, -0.000100, 0.000000, 3.141593, 0.000000],accel_mss,speed_ms,0,blend_radius_m)
    |   movel(p[0.463925, -0.086747, -0.000100, 0.000000, -3.141593, 0.000000],accel_mss,speed_ms,0,blend_radius_m)
    |   movel(p[0.465161, -0.085936, -0.000100, 0.000000, -3.141593, 0.000000],accel_mss,speed_ms,0,blend_radius_m)
    |   movel(p[0.465410, -0.085741, -0.000100, 0.000000, -3.141593, 0.000000],accel_mss,speed_ms,0,0.000)
    |   movel(p[0.465641, -0.085577, -0.000100, 0.000000, -3.141593, 0.000000],accel_mss,speed_ms,0,0.000)
    |   movel(p[0.465838, -0.085451, -0.000100, 0.000000, -3.141593, 0.000000],accel_mss,speed_ms,0,0.000)
    |   movel(p[0.465996, -0.085401, -0.000100, 0.000000, -3.141593, 0.000000],accel_mss,speed_ms,0,0.000)
    |   movel(p[0.466205, -0.085230, -0.000100, 0.000000, -3.141593, 0.000000],accel_mss,speed_ms,0,0.000)
    |   movel(p[0.466448, -0.085012, -0.000100, 0.000000, -3.141593, 0.000000],accel_mss,speed_ms,0,0.000)
    |   movel(p[0.466711, -0.084753, -0.000100, 0.000000, -3.141593, 0.000000],accel_mss,speed_ms,0,0.000)
    |   movel(p[0.466976, -0.084495, -0.000100, 0.000000, -3.141593, 0.000000],accel_mss,speed_ms,0,0.000)
    |   movel(p[0.467224, -0.084277, -0.000100, 0.000000, -3.141593, 0.000000],accel_mss,speed_ms,0,0.000)
    |   movel(p[0.467436, -0.084108, -0.000100, 0.000000, -3.141593, 0.000000],accel_mss,speed_ms,0,0.000)
    |   movel(p[0.467764, -0.083982, -0.000100, 0.000000, -3.141593, 0.000000],accel_mss,speed_ms,0,0.000)
    |   movel(p[0.468845, -0.082916, -0.000100, 0.000000, -3.141593, 0.000000],accel_mss,speed_ms,0,blend_radius_m)
    |   movel(p[0.469914, -0.081837, -0.000100, 0.000000, -3.141593, 0.000000],accel_mss,speed_ms,0,blend_radius_m)
    |   movel(p[0.470011, -0.081601, -0.000100, 0.000000, -3.141593, 0.000000],accel_mss,speed_ms,0,0.000)
    |   movel(p[0.470209, -0.081293, -0.000100, 0.000000, -3.141593, 0.000000],accel_mss,speed_ms,0,0.000)
    |   movel(p[0.470427, -0.081044, -0.000100, 0.000000, -3.141593, 0.000000],accel_mss,speed_ms,0,0.000)
    |   movel(p[0.470686, -0.080778, -0.000100, 0.000000, -3.141593, 0.000000],accel_mss,speed_ms,0,0.000)
    |   movel(p[0.470945, -0.080515, -0.000100, 0.000000, -3.141593, 0.000000],accel_mss,speed_ms,0,0.000)
    |   movel(p[0.471163, -0.080272, -0.000100, 0.000000, -3.141593, 0.000000],accel_mss,speed_ms,0,0.000)
    |   movel(p[0.471334, -0.080064, -0.000100, 0.000000, -3.141593, 0.000000],accel_mss,speed_ms,0,0.000)
    |   movel(p[0.471385, -0.079907, -0.000100, 0.000000, -3.141593, 0.000000],accel_mss,speed_ms,0,0.000)
    |   movel(p[0.471532, -0.079689, -0.000100, 0.000000, -3.141593, 0.000000],accel_mss,speed_ms,0,0.000)
    |   movel(p[0.471719, -0.079434, -0.000100, 0.000000, -3.141593, 0.000000],accel_mss,speed_ms,0,0.000)
    |   movel(p[0.471942, -0.079155, -0.000100, 0.000000, -3.141593, 0.000000],accel_mss,speed_ms,0,0.000)
    |   movel(p[0.472603, -0.078252, -0.000100, 0.000000, -3.141593, 0.000000],accel_mss,speed_ms,0,blend_radius_m)
    |   movel(p[0.473351, -0.077020, -0.000100, 0.000000, -3.141593, 0.000000],accel_mss,speed_ms,0,blend_radius_m)
    |   movel(p[0.474091, -0.075636, -0.000100, 0.000000, 3.141593, 0.000000],accel_mss,speed_ms,0,blend_radius_m)
    |   movel(p[0.474733, -0.074253, -0.000100, 0.000000, -3.141593, 0.000000],accel_mss,speed_ms,0,blend_radius_m)
    |   movel(p[0.474852, -0.073980, -0.000100, 0.000000, 3.141593, 0.000000],accel_mss,speed_ms,0,0.000)
    |   movel(p[0.474997, -0.073653, -0.000100, 0.000000, -3.141593, 0.000000],accel_mss,speed_ms,0,0.000)
    |   movel(p[0.475145, -0.073327, -0.000100, 0.000000, -3.141593, 0.000000],accel_mss,speed_ms,0,0.000)
    |   movel(p[0.475271, -0.073053, -0.000100, 0.000000, -3.141593, 0.000000],accel_mss,speed_ms,0,0.000)
    |   movel(p[0.475382, -0.072802, -0.000100, 0.000000, 3.141593, 0.000000],accel_mss,speed_ms,0,0.000)
    |   movel(p[0.475485, -0.072541, -0.000100, 0.000000, -3.141593, 0.000000],accel_mss,speed_ms,0,0.000)
    |   movel(p[0.475567, -0.072308, -0.000100, 0.000000, -3.141593, 0.000000],accel_mss,speed_ms,0,0.000)
    |   movel(p[0.475606, -0.072153, -0.000100, 0.000000, -3.141593, 0.000000],accel_mss,speed_ms,0,0.000)
    |   movel(p[0.475647, -0.071970, -0.000100, 0.000000, -3.141593, 0.000000],accel_mss,speed_ms,0,0.000)
    |   movel(p[0.475758, -0.071567, -0.000100, 0.000000, -3.141593, 0.000000],accel_mss,speed_ms,0,0.000)
    |   movel(p[0.475895, -0.071089, -0.000100, 0.000000, -3.141593, 0.000000],accel_mss,speed_ms,0,0.000)
    |   movel(p[0.476047, -0.070578, -0.000100, 0.000000, 3.141593, 0.000000],accel_mss,speed_ms,0,blend_radius_m)
    |   movel(p[0.476484, -0.069007, -0.000100, 0.000000, -3.141593, 0.000000],accel_mss,speed_ms,0,blend_radius_m)
    |   movel(p[0.476720, -0.067809, -0.000100, 0.000000, -3.141593, 0.000000],accel_mss,speed_ms,0,blend_radius_m)
    |   movel(p[0.476863, -0.066385, -0.000100, 0.000000, -3.141593, 0.000000],accel_mss,speed_ms,0,blend_radius_m)
    |   movel(p[0.477000, -0.063791, -0.000100, 0.000000, -3.141593, 0.000000],accel_mss,speed_ms,0,blend_radius_m)
    |   movel(p[0.477059, -0.062131, -0.000100, 0.000000, -3.141593, 0.000000],accel_mss,speed_ms,0,blend_radius_m)
    |   movel(p[0.476988, -0.061541, -0.000100, 0.000000, -3.141593, 0.000000],accel_mss,speed_ms,0,blend_radius_m)
    |   movel(p[0.476813, -0.061505, -0.000100, 0.000000, -3.141593, 0.000000],accel_mss,speed_ms,0,0.000)
    |   movel(p[0.476516, -0.061991, -0.000100, 0.000000, -3.141593, 0.000000],accel_mss,speed_ms,0,blend_radius_m)
    |   movel(p[0.476387, -0.062244, -0.000100, 0.000000, 3.141593, 0.000000],accel_mss,speed_ms,0,0.000)
    |   movel(p[0.476214, -0.062542, -0.000100, 0.000000, -3.141593, 0.000000],accel_mss,speed_ms,0,0.000)
    |   movel(p[0.476027, -0.062837, -0.000100, 0.000000, 3.141593, 0.000000],accel_mss,speed_ms,0,0.000)
    |   movel(p[0.475854, -0.063078, -0.000100, 0.000000, 3.141593, 0.000000],accel_mss,speed_ms,0,0.000)
    |   movel(p[0.475691, -0.063307, -0.000100, 0.000000, -3.141593, 0.000000],accel_mss,speed_ms,0,0.000)
    |   movel(p[0.475536, -0.063559, -0.000100, 0.000000, -3.141593, 0.000000],accel_mss,speed_ms,0,0.000)
    |   movel(p[0.475409, -0.063798, -0.000100, 0.000000, -3.141593, 0.000000],accel_mss,speed_ms,0,0.000)
    |   movel(p[0.475338, -0.063978, -0.000100, 0.000000, -3.141593, 0.000000],accel_mss,speed_ms,0,0.000)
    |   movel(p[0.475282, -0.064137, -0.000100, 0.000000, -3.141593, 0.000000],accel_mss,speed_ms,0,0.000)
    |   movel(p[0.475210, -0.064303, -0.000100, 0.000000, -3.141593, 0.000000],accel_mss,speed_ms,0,0.000)
    |   movel(p[0.475132, -0.064453, -0.000100, 0.000000, -3.141593, 0.000000],accel_mss,speed_ms,0,0.000)
    |   movel(p[0.475061, -0.064557, -0.000100, 0.000000, -3.141593, 0.000000],accel_mss,speed_ms,0,0.000)
    |   movel(p[0.474904, -0.064772, -0.000100, 0.000000, -3.141593, 0.000000],accel_mss,speed_ms,0,0.000)
    |   movel(p[0.474722, -0.065062, -0.000100, 0.000000, -3.141593, 0.000000],accel_mss,speed_ms,0,0.000)
    |   movel(p[0.474516, -0.065422, -0.000100, 0.000000, -3.141593, 0.000000],accel_mss,speed_ms,0,0.000)
    |   movel(p[0.474285, -0.065853, -0.000100, 0.000000, -3.141593, 0.000000],accel_mss,speed_ms,0,0.000)
    |   movel(p[0.474175, -0.066058, -0.000100, 0.000000, -3.141593, 0.000000],accel_mss,speed_ms,0,0.000)
    |   movel(p[0.474035, -0.066303, -0.000100, 0.000000, 3.141593, 0.000000],accel_mss,speed_ms,0,0.000)
    |   movel(p[0.473889, -0.066548, -0.000100, 0.000000, -3.141593, 0.000000],accel_mss,speed_ms,0,0.000)
    |   movel(p[0.473761, -0.066753, -0.000100, 0.000000, -3.141593, 0.000000],accel_mss,speed_ms,0,0.000)
    |   movel(p[0.473633, -0.066958, -0.000100, 0.000000, -3.141593, 0.000000],accel_mss,speed_ms,0,0.000)
    |   movel(p[0.473488, -0.067203, -0.000100, 0.000000, -3.141593, 0.000000],accel_mss,speed_ms,0,0.000)
    |   movel(p[0.473350, -0.067449, -0.000100, 0.000000, -3.141593, 0.000000],accel_mss,speed_ms,0,0.000)
    |   movel(p[0.473241, -0.067653, -0.000100, 0.000000, -3.141593, 0.000000],accel_mss,speed_ms,0,0.000)
    |   movel(p[0.473132, -0.067858, -0.000100, 0.000000, -3.141593, 0.000000],accel_mss,speed_ms,0,0.000)
    |   movel(p[0.472993, -0.068103, -0.000100, 0.000000, -3.141593, 0.000000],accel_mss,speed_ms,0,0.000)
    |   movel(p[0.472847, -0.068348, -0.000100, 0.000000, -3.141593, 0.000000],accel_mss,speed_ms,0,0.000)
    |   movel(p[0.472718, -0.068553, -0.000100, 0.000000, -3.141593, 0.000000],accel_mss,speed_ms,0,0.000)
    |   movel(p[0.472587, -0.068763, -0.000100, 0.000000, -3.141593, 0.000000],accel_mss,speed_ms,0,0.000)
    |   movel(p[0.472434, -0.069025, -0.000100, 0.000000, -3.141593, 0.000000],accel_mss,speed_ms,0,0.000)
    |   movel(p[0.472284, -0.069295, -0.000100, 0.000000, -3.141593, 0.000000],accel_mss,speed_ms,0,0.000)
    |   movel(p[0.472162, -0.069528, -0.000100, 0.000000, -3.141593, 0.000000],accel_mss,speed_ms,0,0.000)
    |   movel(p[0.471951, -0.069926, -0.000100, 0.000000, -3.141593, 0.000000],accel_mss,speed_ms,0,0.000)
    |   movel(p[0.471650, -0.070454, -0.000100, 0.000000, -3.141593, 0.000000],accel_mss,speed_ms,0,blend_radius_m)
